QRS_NEXT_CUT()
PTP {E1 34737.351,E2 34737.351}
PTP {X 0,Y 759.916,A -85,B 0,C 180,E1 34737.351,E2 34737.351,E3 0,E4 0,E5 0,E6 0}
QRS_SPEED_INIT()
LIN {X 0,Y 759.916,Z 1215,A -85,B 0,C 180,E1 34737.351,E2 34737.351,E3 0,E4 0,E5 0,E6 0} C_VEL
LIN {X 0,Y 759.916,Z 694.953,A -85,B 0,C 180,E1 34737.351,E2 34737.351} C_VEL
LIN {X 0,Y 759.916,Z 679.951,A -85,B 0,C 180,E1 34737.351,E2 34737.351} C_VEL
LIN {X 0,Y 759.914,Z 679.08,A -85,B 0,C 180,E1 34737.064,E2 34737.064} C_VEL
LIN {X 0,Y 759.912,Z 758.546,A -85,B 0,C 180,E1 34734.185,E2 34734.185} C_VEL
LIN {X 0,Y 759.906,Z 836.117,A -85,B 0,C 180,E1 34731.411,E2 34731.411} C_VEL
LIN {X 0,Y 759.917,Z 950.864,A -85,B 0,C 180,E1 34730.313,E2 34730.313} C_VEL
LIN {X 0,Y 759.912,Z 962.666,A -85,B 0,C 180,E1 34730.113,E2 34730.113} C_VEL
LIN {X 0,Y 759.907,Z 975.52,A -85,B 0,C 180,E1 34729.789,E2 34729.789} C_VEL
LIN {X 0,Y 759.913,Z 990.031,A -85,B 0,C 180,E1 34729.27,E2 34729.27} C_VEL
LIN {X 0,Y 759.899,Z 1001.309,A -85,B 0,C 180,E1 34728.732,E2 34728.732} C_VEL
LIN {X 0,Y 759.919,Z 1011.084,A -85,B 0,C 180,E1 34728.155,E2 34728.155} C_VEL
LIN {X 0,Y 759.915,Z 1020.118,A -85,B 0,C 180,E1 34727.506,E2 34727.506} C_VEL
LIN {X 0,Y 759.915,Z 1028.572,A -85,B 0,C 180,E1 34726.765,E2 34726.765} C_VEL
LIN {X 0,Y 759.911,Z 1037.65,A -85,B 0,C 180,E1 34725.756,E2 34725.756} C_VEL
LIN {X 0,Y 759.916,Z 1043.966,A -85,B 0,C 180,E1 34724.821,E2 34724.821} C_VEL
LIN {X 0,Y 759.916,Z 1048.406,A -85,B 0,C 180,E1 34723.959,E2 34723.959} C_VEL
LIN {X 0,Y 759.912,Z 1051.646,A -85,B 0,C 180,E1 34723.095,E2 34723.095} C_VEL
LIN {X 0,Y 759.918,Z 1053.76,A -85,B 0,C 180,E1 34722.226,E2 34722.226} C_VEL
LIN {X 0,Y 759.907,Z 1054.804,A -85,B 0,C 180,E1 34721.33,E2 34721.33} C_VEL
LIN {X 0,Y 759.913,Z 1054.696,A -85,B 0,C 180,E1 34720.395,E2 34720.395} C_VEL
LIN {X 0,Y 759.905,Z 1052.996,A -85,B 0,C 180,E1 34719.271,E2 34719.271} C_VEL
LIN {X 0,Y 759.917,Z 1049.566,A -85,B 0,C 180,E1 34718.219,E2 34718.219} C_VEL
LIN {X 0,Y 759.908,Z 1045.3,A -85,B 0,C 180,E1 34717.323,E2 34717.323} C_VEL
LIN {X 0,Y 759.913,Z 1040.168,A -85,B 0,C 180,E1 34716.504,E2 34716.504} C_VEL
LIN {X 0,Y 759.917,Z 1034.354,A -85,B 0,C 180,E1 34715.761,E2 34715.761} C_VEL
LIN {X 0,Y 759.919,Z 1027.189,A -85,B 0,C 180,E1 34715.016,E2 34715.016} C_VEL
LIN {X 0,Y 759.916,Z 1019.197,A -85,B 0,C 180,E1 34714.332,E2 34714.332} C_VEL
LIN {X 0,Y 759.919,Z 1009.396,A -85,B 0,C 180,E1 34713.644,E2 34713.644} C_VEL
LIN {X 0,Y 759.904,Z 996.19,A -85,B 0,C 180,E1 34712.917,E2 34712.917} C_VEL
LIN {X 0,Y 759.914,Z 985.016,A -85,B 0,C 180,E1 34712.444,E2 34712.444} C_VEL
LIN {X 0,Y 759.906,Z 973.587,A -85,B 0,C 180,E1 34712.068,E2 34712.068} C_VEL
LIN {X 0,Y 759.914,Z 962.312,A -85,B 0,C 180,E1 34711.79,E2 34711.79} C_VEL
LIN {X 0,Y 759.916,Z 950.123,A -85,B 0,C 180,E1 34711.587,E2 34711.587} C_VEL
LIN {X 0,Y 759.905,Z 835.386,A -85,B 0,C 180,E1 34710.477,E2 34710.477} C_VEL
LIN {X 0,Y 759.917,Z 755.634,A -85,B 0,C 180,E1 34707.62,E2 34707.62} C_VEL
LIN {X 0,Y 759.913,Z 676.623,A -85,B 0,C 180,E1 34704.756,E2 34704.756} C_VEL
LIN {X 0,Y 759.914,Z 596.236,A -85,B 0,C 180,E1 34701.799,E2 34701.799} C_VEL
LIN {X 0,Y 759.89,Z 522.845,A -85,B 0,C 180,E1 34699.051,E2 34699.051} C_VEL
LIN {X 0,Y 759.918,Z 450.182,A -85,B 0,C 180,E1 34696.279,E2 34696.279} C_VEL
LIN {X 0,Y 759.918,Z 393.58,A -85,B 0,C 180,E1 34694.148,E2 34694.148} C_VEL
LIN {X 0,Y 759.86,Z 324.573,A -85,B 0,C 180,E1 34691.632,E2 34691.632} C_VEL
LIN {X 0,Y 759.869,Z 309.663,A -85,B 0,C 180,E1 34691.06,E2 34691.06} C_VEL
LIN {X 0,Y 759.887,Z 319.172,A -85,B 0,C 180,E1 34690.892,E2 34690.892} C_VEL
LIN {X 0,Y 759.917,Z 540.516,A -85,B 0,C 180,E1 34688.23,E2 34688.23} C_VEL
LIN {X 0,Y 759.912,Z 766.77,A -85,B 0,C 180,E1 34685.609,E2 34685.609} C_VEL
LIN {X 0,Y 759.911,Z 803.217,A -85,B 0,C 180,E1 34685.158,E2 34685.158} C_VEL
LIN {X 0,Y 759.908,Z 828.5,A -85,B 0,C 180,E1 34684.704,E2 34684.704} C_VEL
LIN {X 0,Y 759.915,Z 854.556,A -85,B 0,C 180,E1 34684.093,E2 34684.093} C_VEL
LIN {X 0,Y 759.906,Z 879.193,A -85,B 0,C 180,E1 34683.368,E2 34683.368} C_VEL
LIN {X 0,Y 759.918,Z 906.079,A -85,B 0,C 180,E1 34682.425,E2 34682.425} C_VEL
LIN {X 0,Y 759.915,Z 928.461,A -85,B 0,C 180,E1 34681.5,E2 34681.5} C_VEL
LIN {X 0,Y 759.914,Z 947.581,A -85,B 0,C 180,E1 34680.612,E2 34680.612} C_VEL
LIN {X 0,Y 759.914,Z 966.174,A -85,B 0,C 180,E1 34679.653,E2 34679.653} C_VEL
LIN {X 0,Y 759.91,Z 985.832,A -85,B 0,C 180,E1 34678.532,E2 34678.532} C_VEL
LIN {X 0,Y 759.91,Z 1009.761,A -85,B 0,C 180,E1 34676.998,E2 34676.998} C_VEL
LIN {X 0,Y 759.915,Z 1028.449,A -85,B 0,C 180,E1 34675.652,E2 34675.652} C_VEL
LIN {X 0,Y 759.893,Z 1047.319,A -85,B 0,C 180,E1 34674.157,E2 34674.157} C_VEL
LIN {X 0,Y 759.911,Z 1066.636,A -85,B 0,C 180,E1 34672.432,E2 34672.432} C_VEL
LIN {X 0,Y 759.897,Z 1081.386,A -85,B 0,C 180,E1 34670.972,E2 34670.972} C_VEL
LIN {X 0,Y 759.909,Z 1095.388,A -85,B 0,C 180,E1 34669.445,E2 34669.445} C_VEL
LIN {X 0,Y 759.911,Z 1111.611,A -85,B 0,C 180,E1 34667.454,E2 34667.454} C_VEL
LIN {X 0,Y 759.891,Z 1123.379,A -85,B 0,C 180,E1 34665.806,E2 34665.806} C_VEL
LIN {X 0,Y 759.916,Z 1133.313,A -85,B 0,C 180,E1 34664.245,E2 34664.245} C_VEL
LIN {X 0,Y 759.917,Z 1142.044,A -85,B 0,C 180,E1 34662.694,E2 34662.694} C_VEL
LIN {X 0,Y 759.898,Z 1149.999,A -85,B 0,C 180,E1 34661.077,E2 34661.077} C_VEL
LIN {X 0,Y 759.918,Z 1157.72,A -85,B 0,C 180,E1 34659.238,E2 34659.238} C_VEL
LIN {X 0,Y 759.912,Z 1164.34,A -85,B 0,C 180,E1 34657.258,E2 34657.258} C_VEL
LIN {X 0,Y 759.91,Z 1169.506,A -85,B 0,C 180,E1 34655.21,E2 34655.21} C_VEL
LIN {X 0,Y 759.912,Z 1173.032,A -85,B 0,C 180,E1 34653.093,E2 34653.093} C_VEL
LIN {X 0,Y 759.908,Z 1174.635,A -85,B 0,C 180,E1 34651.207,E2 34651.207} C_VEL
LIN {X 0,Y 759.89,Z 1174.841,A -85,B 0,C 180,E1 34649.398,E2 34649.398} C_VEL
LIN {X 0,Y 759.905,Z 1173.876,A -85,B 0,C 180,E1 34647.588,E2 34647.588} C_VEL
LIN {X 0,Y 759.906,Z 1171.005,A -85,B 0,C 180,E1 34645.473,E2 34645.473} C_VEL
LIN {X 0,Y 759.91,Z 1166.488,A -85,B 0,C 180,E1 34643.428,E2 34643.428} C_VEL
LIN {X 0,Y 759.917,Z 1160.522,A -85,B 0,C 180,E1 34641.45,E2 34641.45} C_VEL
LIN {X 0,Y 759.892,Z 1152.552,A -85,B 0,C 180,E1 34639.386,E2 34639.386} C_VEL
LIN {X 0,Y 759.913,Z 1142.943,A -85,B 0,C 180,E1 34637.385,E2 34637.385} C_VEL
LIN {X 0,Y 759.918,Z 1133.863,A -85,B 0,C 180,E1 34635.757,E2 34635.757} C_VEL
LIN {X 0,Y 759.897,Z 1124.515,A -85,B 0,C 180,E1 34634.274,E2 34634.274} C_VEL
LIN {X 0,Y 759.896,Z 1114.001,A -85,B 0,C 180,E1 34632.78,E2 34632.78} C_VEL
LIN {X 0,Y 759.906,Z 1101.586,A -85,B 0,C 180,E1 34631.195,E2 34631.195} C_VEL
LIN {X 0,Y 759.904,Z 1084.615,A -85,B 0,C 180,E1 34629.272,E2 34629.272} C_VEL
LIN {X 0,Y 759.894,Z 1069.306,A -85,B 0,C 180,E1 34627.732,E2 34627.732} C_VEL
LIN {X 0,Y 759.911,Z 1053.867,A -85,B 0,C 180,E1 34626.32,E2 34626.32} C_VEL
LIN {X 0,Y 759.9,Z 1033.545,A -85,B 0,C 180,E1 34624.642,E2 34624.642} C_VEL
LIN {X 0,Y 759.916,Z 1014.708,A -85,B 0,C 180,E1 34623.258,E2 34623.258} C_VEL
LIN {X 0,Y 759.901,Z 995.825,A -85,B 0,C 180,E1 34621.996,E2 34621.996} C_VEL
LIN {X 0,Y 759.904,Z 972.23,A -85,B 0,C 180,E1 34620.583,E2 34620.583} C_VEL
LIN {X 0,Y 759.915,Z 950.344,A -85,B 0,C 180,E1 34619.434,E2 34619.434} C_VEL
LIN {X 0,Y 759.912,Z 931.714,A -85,B 0,C 180,E1 34618.554,E2 34618.554} C_VEL
LIN {X 0,Y 759.919,Z 912.668,A -85,B 0,C 180,E1 34617.748,E2 34617.748} C_VEL
LIN {X 0,Y 759.92,Z 893.868,A -85,B 0,C 180,E1 34617.04,E2 34617.04} C_VEL
LIN {X 0,Y 759.909,Z 875.428,A -85,B 0,C 180,E1 34616.426,E2 34616.426} C_VEL
LIN {X 0,Y 759.912,Z 852.836,A -85,B 0,C 180,E1 34615.773,E2 34615.773} C_VEL
LIN {X 0,Y 759.914,Z 826.079,A -85,B 0,C 180,E1 34615.155,E2 34615.155} C_VEL
LIN {X 0,Y 759.91,Z 799.971,A -85,B 0,C 180,E1 34614.705,E2 34614.705} C_VEL
LIN {X 0,Y 759.919,Z 744.192,A -85,B 0,C 180,E1 34614.044,E2 34614.044} C_VEL
LIN {X 0,Y 759.912,Z 520.251,A -85,B 0,C 180,E1 34611.44,E2 34611.44} C_VEL
LIN {X 0,Y 759.881,Z 320.944,A -85,B 0,C 180,E1 34609.038,E2 34609.038} C_VEL
LIN {X 0,Y 759.906,Z 309.576,A -85,B 0,C 180,E1 34608.251,E2 34608.251} C_VEL
LIN {X 0,Y 759.906,Z 309.576,A -85,B 0,C 180,E1 34605.257,E2 34605.257} C_VEL
LIN {X 0,Y 759.897,Z 309.577,A -85,B 0,C 180,E1 34602.426,E2 34602.426} C_VEL
LIN {X 0,Y 759.915,Z 309.575,A -85,B 0,C 180,E1 34599.362,E2 34599.362} C_VEL
LIN {X 0,Y 759.895,Z 309.577,A -85,B 0,C 180,E1 34596.589,E2 34596.589} C_VEL
LIN {X 0,Y 759.894,Z 309.575,A -85,B 0,C 180,E1 34593.73,E2 34593.73} C_VEL
LIN {X 0,Y 759.909,Z 309.577,A -85,B 0,C 180,E1 34590.875,E2 34590.875} C_VEL
LIN {X 0,Y 759.88,Z 309.577,A -85,B 0,C 180,E1 34588.104,E2 34588.104} C_VEL
LIN {X 0,Y 759.916,Z 309.575,A -85,B 0,C 180,E1 34585.234,E2 34585.234} C_VEL
LIN {X 0,Y 759.888,Z 309.577,A -85,B 0,C 180,E1 34582.433,E2 34582.433} C_VEL
LIN {X 0,Y 759.881,Z 309.576,A -85,B 0,C 180,E1 34579.766,E2 34579.766} C_VEL
LIN {X 0,Y 759.919,Z 309.577,A -85,B 0,C 180,E1 34576.905,E2 34576.905} C_VEL
LIN {X 0,Y 759.88,Z 309.577,A -85,B 0,C 180,E1 34574.012,E2 34574.012} C_VEL
LIN {X 0,Y 759.899,Z 309.577,A -85,B 0,C 180,E1 34571.23,E2 34571.23} C_VEL
LIN {X 0,Y 759.889,Z 309.577,A -85,B 0,C 180,E1 34568.399,E2 34568.399} C_VEL
LIN {X 0,Y 759.884,Z 309.576,A -85,B 0,C 180,E1 34565.588,E2 34565.588} C_VEL
LIN {X 0,Y 759.919,Z 309.576,A -85,B 0,C 180,E1 34562.791,E2 34562.791} C_VEL
LIN {X 0,Y 759.881,Z 309.577,A -85,B 0,C 180,E1 34559.849,E2 34559.849} C_VEL
LIN {X 0,Y 759.913,Z 309.576,A -85,B 0,C 180,E1 34557.03,E2 34557.03} C_VEL
LIN {X 0,Y 759.903,Z 309.574,A -85,B 0,C 180,E1 34554.109,E2 34554.109} C_VEL
LIN {X 0,Y 759.91,Z 309.578,A -85,B 0,C 180,E1 34551.144,E2 34551.144} C_VEL
LIN {X 0,Y 759.916,Z 309.572,A -85,B 0,C 180,E1 34548.155,E2 34548.155} C_VEL
LIN {X 0,Y 759.912,Z 309.576,A -85,B 0,C 180,E1 34545.211,E2 34545.211} C_VEL
LIN {X 0,Y 759.898,Z 309.574,A -85,B 0,C 180,E1 34542.293,E2 34542.293} C_VEL
LIN {X 0,Y 759.917,Z 309.575,A -85,B 0,C 180,E1 34539.432,E2 34539.432} C_VEL
LIN {X 0,Y 759.882,Z 309.576,A -85,B 0,C 180,E1 34536.605,E2 34536.605} C_VEL
LIN {X 0,Y 759.905,Z 337.086,A -85,B 0,C 180,E1 34534.557,E2 34534.557} C_VEL
LIN {X 0,Y 759.898,Z 371.805,A -85,B 0,C 180,E1 34532.11,E2 34532.11} C_VEL
LIN {X 0,Y 759.915,Z 409.049,A -85,B 0,C 180,E1 34529.607,E2 34529.607} C_VEL
LIN {X 0,Y 759.914,Z 451.966,A -85,B 0,C 180,E1 34526.858,E2 34526.858} C_VEL
LIN {X 0,Y 759.917,Z 494.443,A -85,B 0,C 180,E1 34524.253,E2 34524.253} C_VEL
LIN {X 0,Y 759.917,Z 511.943,A -85,B 0,C 180,E1 34523.177,E2 34523.177} C_VEL
LIN {X 0,Y 759.868,Z 518.357,A -85,B 0,C 180,E1 34522.632,E2 34522.632} C_VEL
LIN {X 0,Y 759.872,Z 521.733,A -85,B 0,C 180,E1 34522.179,E2 34522.179} C_VEL
LIN {X 0,Y 759.916,Z 522.967,A -85,B 0,C 180,E1 34521.767,E2 34521.767} C_VEL
LIN {X 0,Y 759.913,Z 522.331,A -85,B 0,C 180,E1 34521.414,E2 34521.414} C_VEL
LIN {X 0,Y 759.893,Z 519.98,A -85,B 0,C 180,E1 34521.123,E2 34521.123} C_VEL
LIN {X 0,Y 759.887,Z 515.523,A -85,B 0,C 180,E1 34520.878,E2 34520.878} C_VEL
LIN {X 0,Y 759.891,Z 508.959,A -85,B 0,C 180,E1 34520.71,E2 34520.71} C_VEL
LIN {X 0,Y 759.895,Z 499.107,A -85,B 0,C 180,E1 34520.633,E2 34520.633} C_VEL
LIN {X 0,Y 759.896,Z 309.577,A -85,B 0,C 180,E1 34520.619,E2 34520.619} C_VEL
LIN {X 0,Y 759.885,Z 309.578,A -85,B 0,C 180,E1 34517.849,E2 34517.849} C_VEL
LIN {X 0,Y 759.914,Z 309.575,A -85,B 0,C 180,E1 34515.042,E2 34515.042} C_VEL
LIN {X 0,Y 759.901,Z 309.831,A -85,B 0,C 180,E1 34513.53,E2 34513.53} C_VEL
LIN {X 0,Y 759.904,Z 350.586,A -85,B 0,C 180,E1 34510.919,E2 34510.919} C_VEL
LIN {X 0,Y 759.912,Z 566.45,A -85,B 0,C 180,E1 34508.323,E2 34508.323} C_VEL
LIN {X 0,Y 759.917,Z 792.192,A -85,B 0,C 180,E1 34505.706,E2 34505.706} C_VEL
LIN {X 0,Y 759.911,Z 831.842,A -85,B 0,C 180,E1 34505.223,E2 34505.223} C_VEL
LIN {X 0,Y 759.908,Z 857.533,A -85,B 0,C 180,E1 34504.769,E2 34504.769} C_VEL
LIN {X 0,Y 759.913,Z 884.387,A -85,B 0,C 180,E1 34504.143,E2 34504.143} C_VEL
LIN {X 0,Y 759.907,Z 909.999,A -85,B 0,C 180,E1 34503.388,E2 34503.388} C_VEL
LIN {X 0,Y 759.918,Z 937.266,A -85,B 0,C 180,E1 34502.422,E2 34502.422} C_VEL
LIN {X 0,Y 759.915,Z 958.597,A -85,B 0,C 180,E1 34501.539,E2 34501.539} C_VEL
LIN {X 0,Y 759.912,Z 977.517,A -85,B 0,C 180,E1 34500.66,E2 34500.66} C_VEL
LIN {X 0,Y 759.912,Z 996.378,A -85,B 0,C 180,E1 34499.687,E2 34499.687} C_VEL
LIN {X 0,Y 759.903,Z 1015.171,A -85,B 0,C 180,E1 34498.616,E2 34498.616} C_VEL
LIN {X 0,Y 759.901,Z 1038.015,A -85,B 0,C 180,E1 34497.166,E2 34497.166} C_VEL
LIN {X 0,Y 759.916,Z 1057.965,A -85,B 0,C 180,E1 34495.734,E2 34495.734} C_VEL
LIN {X 0,Y 759.902,Z 1075.357,A -85,B 0,C 180,E1 34494.361,E2 34494.361} C_VEL
LIN {X 0,Y 759.914,Z 1095.42,A -85,B 0,C 180,E1 34492.593,E2 34492.593} C_VEL
LIN {X 0,Y 759.892,Z 1110.551,A -85,B 0,C 180,E1 34491.104,E2 34491.104} C_VEL
LIN {X 0,Y 759.911,Z 1124.385,A -85,B 0,C 180,E1 34489.603,E2 34489.603} C_VEL
LIN {X 0,Y 759.914,Z 1139.588,A -85,B 0,C 180,E1 34487.773,E2 34487.773} C_VEL
LIN {X 0,Y 759.889,Z 1152.649,A -85,B 0,C 180,E1 34485.961,E2 34485.961} C_VEL
LIN {X 0,Y 759.91,Z 1162.664,A -85,B 0,C 180,E1 34484.399,E2 34484.399} C_VEL
LIN {X 0,Y 759.914,Z 1171.531,A -85,B 0,C 180,E1 34482.836,E2 34482.836} C_VEL
LIN {X 0,Y 759.915,Z 1179.146,A -85,B 0,C 180,E1 34481.305,E2 34481.305} C_VEL
LIN {X 0,Y 759.906,Z 1186.727,A -85,B 0,C 180,E1 34479.542,E2 34479.542} C_VEL
LIN {X 0,Y 759.908,Z 1193.596,A -85,B 0,C 180,E1 34477.56,E2 34477.56} C_VEL
LIN {X 0,Y 759.91,Z 1199.11,A -85,B 0,C 180,E1 34475.435,E2 34475.435} C_VEL
LIN {X 0,Y 759.916,Z 1202.587,A -85,B 0,C 180,E1 34473.469,E2 34473.469} C_VEL
LIN {X 0,Y 759.914,Z 1204.581,A -85,B 0,C 180,E1 34471.432,E2 34471.432} C_VEL
LIN {X 0,Y 759.889,Z 1204.849,A -85,B 0,C 180,E1 34469.471,E2 34469.471} C_VEL
LIN {X 0,Y 759.907,Z 1203.906,A -85,B 0,C 180,E1 34467.661,E2 34467.661} C_VEL
LIN {X 0,Y 759.908,Z 1201.052,A -85,B 0,C 180,E1 34465.547,E2 34465.547} C_VEL
LIN {X 0,Y 759.914,Z 1196.563,A -85,B 0,C 180,E1 34463.502,E2 34463.502} C_VEL
LIN {X 0,Y 759.912,Z 1190.625,A -85,B 0,C 180,E1 34461.525,E2 34461.525} C_VEL
LIN {X 0,Y 759.896,Z 1182.676,A -85,B 0,C 180,E1 34459.461,E2 34459.461} C_VEL
LIN {X 0,Y 759.905,Z 1173.105,A -85,B 0,C 180,E1 34457.46,E2 34457.46} C_VEL
LIN {X 0,Y 759.91,Z 1164.049,A -85,B 0,C 180,E1 34455.833,E2 34455.833} C_VEL
LIN {X 0,Y 759.894,Z 1154.204,A -85,B 0,C 180,E1 34454.272,E2 34454.272} C_VEL
LIN {X 0,Y 759.904,Z 1143.658,A -85,B 0,C 180,E1 34452.778,E2 34452.778} C_VEL
LIN {X 0,Y 759.896,Z 1129.919,A -85,B 0,C 180,E1 34451.033,E2 34451.033} C_VEL
LIN {X 0,Y 759.898,Z 1113.38,A -85,B 0,C 180,E1 34449.189,E2 34449.189} C_VEL
LIN {X 0,Y 759.898,Z 1098.813,A -85,B 0,C 180,E1 34447.73,E2 34447.73} C_VEL
LIN {X 0,Y 759.911,Z 1082.64,A -85,B 0,C 180,E1 34446.256,E2 34446.256} C_VEL
LIN {X 0,Y 759.91,Z 1061.259,A -85,B 0,C 180,E1 34444.515,E2 34444.515} C_VEL
LIN {X 0,Y 759.909,Z 1043.428,A -85,B 0,C 180,E1 34443.213,E2 34443.213} C_VEL
LIN {X 0,Y 759.914,Z 1024.236,A -85,B 0,C 180,E1 34441.939,E2 34441.939} C_VEL
LIN {X 0,Y 759.906,Z 999.416,A -85,B 0,C 180,E1 34440.477,E2 34440.477} C_VEL
LIN {X 0,Y 759.913,Z 979.389,A -85,B 0,C 180,E1 34439.432,E2 34439.432} C_VEL
LIN {X 0,Y 759.912,Z 960.652,A -85,B 0,C 180,E1 34438.552,E2 34438.552} C_VEL
LIN {X 0,Y 759.918,Z 941.519,A -85,B 0,C 180,E1 34437.747,E2 34437.747} C_VEL
LIN {X 0,Y 759.92,Z 922.548,A -85,B 0,C 180,E1 34437.038,E2 34437.038} C_VEL
LIN {X 0,Y 759.91,Z 903.935,A -85,B 0,C 180,E1 34436.425,E2 34436.425} C_VEL
LIN {X 0,Y 759.914,Z 881.874,A -85,B 0,C 180,E1 34435.793,E2 34435.793} C_VEL
LIN {X 0,Y 759.909,Z 855.665,A -85,B 0,C 180,E1 34435.192,E2 34435.192} C_VEL
LIN {X 0,Y 759.91,Z 828.993,A -85,B 0,C 180,E1 34434.735,E2 34434.735} C_VEL
LIN {X 0,Y 759.914,Z 731.51,A -85,B 0,C 180,E1 34433.599,E2 34433.599} C_VEL
LIN {X 0,Y 759.915,Z 508.586,A -85,B 0,C 180,E1 34430.991,E2 34430.991} C_VEL
LIN {X 0,Y 759.916,Z 343.629,A -85,B 0,C 180,E1 34428.982,E2 34428.982} C_VEL
LIN {X 0,Y 759.896,Z 309.576,A -85,B 0,C 180,E1 34428.331,E2 34428.331} C_VEL
LIN {X 0,Y 759.903,Z 309.578,A -85,B 0,C 180,E1 34425.494,E2 34425.494} C_VEL
LIN {X 0,Y 759.909,Z 309.577,A -85,B 0,C 180,E1 34422.647,E2 34422.647} C_VEL
LIN {X 0,Y 759.877,Z 309.577,A -85,B 0,C 180,E1 34419.784,E2 34419.784} C_VEL
LIN {X 0,Y 759.883,Z 309.574,A -85,B 0,C 180,E1 34417.061,E2 34417.061} C_VEL
LIN {X 0,Y 759.907,Z 309.575,A -85,B 0,C 180,E1 34414.093,E2 34414.093} C_VEL
LIN {X 0,Y 759.918,Z 309.575,A -85,B 0,C 180,E1 34411.211,E2 34411.211} C_VEL
LIN {X 0,Y 759.919,Z 309.573,A -85,B 0,C 180,E1 34408.274,E2 34408.274} C_VEL
LIN {X 0,Y 759.873,Z 309.575,A -85,B 0,C 180,E1 34405.311,E2 34405.311} C_VEL
LIN {X 0,Y 759.875,Z 309.577,A -85,B 0,C 180,E1 34402.678,E2 34402.678} C_VEL
LIN {X 0,Y 759.914,Z 309.574,A -85,B 0,C 180,E1 34399.815,E2 34399.815} C_VEL
LIN {X 0,Y 759.907,Z 309.577,A -85,B 0,C 180,E1 34396.944,E2 34396.944} C_VEL
LIN {X 0,Y 759.913,Z 309.573,A -85,B 0,C 180,E1 34394.011,E2 34394.011} C_VEL
LIN {X 0,Y 759.881,Z 309.577,A -85,B 0,C 180,E1 34390.999,E2 34390.999} C_VEL
LIN {X 0,Y 759.916,Z 309.801,A -85,B 0,C 180,E1 34390.594,E2 34390.594} C_VEL
LIN {X 0,Y 759.917,Z 389.194,A -85,B 0,C 180,E1 34387.865,E2 34387.865} C_VEL
LIN {X 0,Y 759.904,Z 437.584,A -85,B 0,C 180,E1 34386.118,E2 34386.118} C_VEL
LIN {X 0,Y 759.914,Z 512.66,A -85,B 0,C 180,E1 34383.243,E2 34383.243} C_VEL
LIN {X 0,Y 759.891,Z 587.07,A -85,B 0,C 180,E1 34380.452,E2 34380.452} C_VEL
LIN {X 0,Y 759.911,Z 661.684,A -85,B 0,C 180,E1 34377.7,E2 34377.7} C_VEL
LIN {X 0,Y 759.914,Z 679.08,A -85,B 0,C 180,E1 34377.064,E2 34377.064} C_VEL
LIN {X 0,Y 758.952,Z 686.122,A -85,B 0,C 180,E1 34376.828,E2 34376.828} C_VEL
LIN {X 0,Y 752.87,Z 705.08,A -85,B 0,C 180,E1 34376.263,E2 34376.263} C_VEL
LIN {X 0,Y 752.141,Z 711.123,A -85,B 0,C 180,E1 34376.057,E2 34376.057} C_VEL
LIN {X 0,Y 752.048,Z 789.43,A -85,B 0,C 180,E1 34373.204,E2 34373.204} C_VEL
LIN {X 0,Y 752.039,Z 836.739,A -85,B 0,C 180,E1 34371.516,E2 34371.516} C_VEL
LIN {X 0,Y 752.023,Z 951.389,A -85,B 0,C 180,E1 34370.406,E2 34370.406} C_VEL
LIN {X 0,Y 752.007,Z 965.681,A -85,B 0,C 180,E1 34370.149,E2 34370.149} C_VEL
LIN {X 0,Y 751.99,Z 980.545,A -85,B 0,C 180,E1 34369.72,E2 34369.72} C_VEL
LIN {X 0,Y 751.975,Z 992.811,A -85,B 0,C 180,E1 34369.233,E2 34369.233} C_VEL
LIN {X 0,Y 751.954,Z 1003.593,A -85,B 0,C 180,E1 34368.689,E2 34368.689} C_VEL
LIN {X 0,Y 751.952,Z 1014.743,A -85,B 0,C 180,E1 34367.989,E2 34367.989} C_VEL
LIN {X 0,Y 751.934,Z 1024.967,A -85,B 0,C 180,E1 34367.169,E2 34367.169} C_VEL
LIN {X 0,Y 751.928,Z 1033.456,A -85,B 0,C 180,E1 34366.308,E2 34366.308} C_VEL
LIN {X 0,Y 751.922,Z 1039.959,A -85,B 0,C 180,E1 34365.485,E2 34365.485} C_VEL
LIN {X 0,Y 751.912,Z 1045.589,A -85,B 0,C 180,E1 34364.576,E2 34364.576} C_VEL
LIN {X 0,Y 751.912,Z 1050.595,A -85,B 0,C 180,E1 34363.466,E2 34363.466} C_VEL
LIN {X 0,Y 751.915,Z 1053.568,A -85,B 0,C 180,E1 34362.35,E2 34362.35} C_VEL
LIN {X 0,Y 751.908,Z 1054.774,A -85,B 0,C 180,E1 34361.388,E2 34361.388} C_VEL
LIN {X 0,Y 751.912,Z 1054.715,A -85,B 0,C 180,E1 34360.421,E2 34360.421} C_VEL
LIN {X 0,Y 751.906,Z 1053.069,A -85,B 0,C 180,E1 34359.284,E2 34359.284} C_VEL
LIN {X 0,Y 751.917,Z 1049.358,A -85,B 0,C 180,E1 34358.14,E2 34358.14} C_VEL
LIN {X 0,Y 751.913,Z 1045.023,A -85,B 0,C 180,E1 34357.234,E2 34357.234} C_VEL
LIN {X 0,Y 751.923,Z 1039.63,A -85,B 0,C 180,E1 34356.379,E2 34356.379} C_VEL
LIN {X 0,Y 751.926,Z 1033.188,A -85,B 0,C 180,E1 34355.571,E2 34355.571} C_VEL
LIN {X 0,Y 751.939,Z 1024.748,A -85,B 0,C 180,E1 34354.72,E2 34354.72} C_VEL
LIN {X 0,Y 751.955,Z 1013.524,A -85,B 0,C 180,E1 34353.84,E2 34353.84} C_VEL
LIN {X 0,Y 751.951,Z 1003.326,A -85,B 0,C 180,E1 34353.206,E2 34353.206} C_VEL
LIN {X 0,Y 751.976,Z 992.248,A -85,B 0,C 180,E1 34352.652,E2 34352.652} C_VEL
LIN {X 0,Y 751.987,Z 979.149,A -85,B 0,C 180,E1 34352.14,E2 34352.14} C_VEL
LIN {X 0,Y 752.01,Z 963.946,A -85,B 0,C 180,E1 34351.726,E2 34351.726} C_VEL
LIN {X 0,Y 752.022,Z 950.66,A -85,B 0,C 180,E1 34351.494,E2 34351.494} C_VEL
LIN {X 0,Y 752.016,Z 835.782,A -85,B 0,C 180,E1 34350.38,E2 34350.38} C_VEL
LIN {X 0,Y 752.096,Z 755.202,A -85,B 0,C 180,E1 34347.463,E2 34347.463} C_VEL
LIN {X 0,Y 752.178,Z 675.878,A -85,B 0,C 180,E1 34344.557,E2 34344.557} C_VEL
LIN {X 0,Y 752.281,Z 596.524,A -85,B 0,C 180,E1 34341.607,E2 34341.607} C_VEL
LIN {X 0,Y 752.373,Z 521.834,A -85,B 0,C 180,E1 34338.782,E2 34338.782} C_VEL
LIN {X 0,Y 752.428,Z 453.896,A -85,B 0,C 180,E1 34336.183,E2 34336.183} C_VEL
LIN {X 0,Y 752.292,Z 406.665,A -85,B 0,C 180,E1 34334.414,E2 34334.414} C_VEL
LIN {X 0,Y 752.341,Z 331.817,A -85,B 0,C 180,E1 34331.675,E2 34331.675} C_VEL
LIN {X 0,Y 752.372,Z 323.165,A -85,B 0,C 180,E1 34331.341,E2 34331.341} C_VEL
LIN {X 0,Y 753.749,Z 325.279,A -85,B 0,C 180,E1 34331.222,E2 34331.222} C_VEL
LIN {X 0,Y 753.655,Z 505.38,A -85,B 0,C 180,E1 34329.028,E2 34329.028} C_VEL
LIN {X 0,Y 753.438,Z 733.72,A -85,B 0,C 180,E1 34326.345,E2 34326.345} C_VEL
LIN {X 0,Y 753.352,Z 799.65,A -85,B 0,C 180,E1 34325.563,E2 34325.563} C_VEL
LIN {X 0,Y 753.277,Z 826.497,A -85,B 0,C 180,E1 34325.098,E2 34325.098} C_VEL
LIN {X 0,Y 753.193,Z 854.407,A -85,B 0,C 180,E1 34324.444,E2 34324.444} C_VEL
LIN {X 0,Y 753.094,Z 878.412,A -85,B 0,C 180,E1 34323.735,E2 34323.735} C_VEL
LIN {X 0,Y 752.988,Z 903.865,A -85,B 0,C 180,E1 34322.851,E2 34322.851} C_VEL
LIN {X 0,Y 752.861,Z 927.675,A -85,B 0,C 180,E1 34321.866,E2 34321.866} C_VEL
LIN {X 0,Y 752.761,Z 947.599,A -85,B 0,C 180,E1 34320.935,E2 34320.935} C_VEL
LIN {X 0,Y 752.666,Z 966.993,A -85,B 0,C 180,E1 34319.924,E2 34319.924} C_VEL
LIN {X 0,Y 752.563,Z 987.659,A -85,B 0,C 180,E1 34318.728,E2 34318.728} C_VEL
LIN {X 0,Y 752.423,Z 1010.984,A -85,B 0,C 180,E1 34317.203,E2 34317.203} C_VEL
LIN {X 0,Y 752.347,Z 1029.569,A -85,B 0,C 180,E1 34315.845,E2 34315.845} C_VEL
LIN {X 0,Y 752.234,Z 1049.49,A -85,B 0,C 180,E1 34314.237,E2 34314.237} C_VEL
LIN {X 0,Y 752.171,Z 1067.498,A -85,B 0,C 180,E1 34312.593,E2 34312.593} C_VEL
LIN {X 0,Y 752.096,Z 1082.173,A -85,B 0,C 180,E1 34311.118,E2 34311.118} C_VEL
LIN {X 0,Y 752.054,Z 1098.235,A -85,B 0,C 180,E1 34309.334,E2 34309.334} C_VEL
LIN {X 0,Y 752.003,Z 1112.745,A -85,B 0,C 180,E1 34307.488,E2 34307.488} C_VEL
LIN {X 0,Y 751.955,Z 1123.417,A -85,B 0,C 180,E1 34305.973,E2 34305.973} C_VEL
LIN {X 0,Y 751.959,Z 1133.317,A -85,B 0,C 180,E1 34304.399,E2 34304.399} C_VEL
LIN {X 0,Y 751.932,Z 1142.047,A -85,B 0,C 180,E1 34302.831,E2 34302.831} C_VEL
LIN {X 0,Y 751.923,Z 1150.002,A -85,B 0,C 180,E1 34301.196,E2 34301.196} C_VEL
LIN {X 0,Y 751.926,Z 1158.014,A -85,B 0,C 180,E1 34299.26,E2 34299.26} C_VEL
LIN {X 0,Y 751.916,Z 1164.617,A -85,B 0,C 180,E1 34297.239,E2 34297.239} C_VEL
LIN {X 0,Y 751.907,Z 1169.505,A -85,B 0,C 180,E1 34295.266,E2 34295.266} C_VEL
LIN {X 0,Y 751.911,Z 1172.929,A -85,B 0,C 180,E1 34293.203,E2 34293.203} C_VEL
LIN {X 0,Y 751.911,Z 1174.615,A -85,B 0,C 180,E1 34291.296,E2 34291.296} C_VEL
LIN {X 0,Y 751.889,Z 1174.866,A -85,B 0,C 180,E1 34289.468,E2 34289.468} C_VEL
LIN {X 0,Y 751.907,Z 1173.955,A -85,B 0,C 180,E1 34287.638,E2 34287.638} C_VEL
LIN {X 0,Y 751.908,Z 1171.13,A -85,B 0,C 180,E1 34285.501,E2 34285.501} C_VEL
LIN {X 0,Y 751.917,Z 1166.876,A -85,B 0,C 180,E1 34283.511,E2 34283.511} C_VEL
LIN {X 0,Y 751.924,Z 1160.79,A -85,B 0,C 180,E1 34281.436,E2 34281.436} C_VEL
LIN {X 0,Y 751.905,Z 1152.822,A -85,B 0,C 180,E1 34279.338,E2 34279.338} C_VEL
LIN {X 0,Y 751.941,Z 1143.351,A -85,B 0,C 180,E1 34277.327,E2 34277.327} C_VEL
LIN {X 0,Y 751.961,Z 1134.326,A -85,B 0,C 180,E1 34275.682,E2 34275.682} C_VEL
LIN {X 0,Y 751.956,Z 1124.511,A -85,B 0,C 180,E1 34274.103,E2 34274.103} C_VEL
LIN {X 0,Y 751.997,Z 1113.998,A -85,B 0,C 180,E1 34272.593,E2 34272.593} C_VEL
LIN {X 0,Y 752.031,Z 1101.583,A -85,B 0,C 180,E1 34270.99,E2 34270.99} C_VEL
LIN {X 0,Y 752.09,Z 1084.612,A -85,B 0,C 180,E1 34269.047,E2 34269.047} C_VEL
LIN {X 0,Y 752.152,Z 1069.304,A -85,B 0,C 180,E1 34267.491,E2 34267.491} C_VEL
LIN {X 0,Y 752.21,Z 1052.646,A -85,B 0,C 180,E1 34265.953,E2 34265.953} C_VEL
LIN {X 0,Y 752.343,Z 1031.328,A -85,B 0,C 180,E1 34264.2,E2 34264.2} C_VEL
LIN {X 0,Y 752.415,Z 1012.89,A -85,B 0,C 180,E1 34262.841,E2 34262.841} C_VEL
LIN {X 0,Y 752.546,Z 990.973,A -85,B 0,C 180,E1 34261.382,E2 34261.382} C_VEL
LIN {X 0,Y 752.657,Z 968.678,A -85,B 0,C 180,E1 34260.078,E2 34260.078} C_VEL
LIN {X 0,Y 752.758,Z 949.448,A -85,B 0,C 180,E1 34259.067,E2 34259.067} C_VEL
LIN {X 0,Y 752.853,Z 929.72,A -85,B 0,C 180,E1 34258.136,E2 34258.136} C_VEL
LIN {X 0,Y 752.951,Z 909.498,A -85,B 0,C 180,E1 34257.285,E2 34257.285} C_VEL
LIN {X 0,Y 753.076,Z 884.196,A -85,B 0,C 180,E1 34256.356,E2 34256.356} C_VEL
LIN {X 0,Y 753.178,Z 856.109,A -85,B 0,C 180,E1 34255.512,E2 34255.512} C_VEL
LIN {X 0,Y 753.274,Z 830.147,A -85,B 0,C 180,E1 34254.89,E2 34254.89} C_VEL
LIN {X 0,Y 753.349,Z 803.571,A -85,B 0,C 180,E1 34254.404,E2 34254.404} C_VEL
LIN {X 0,Y 753.404,Z 766.162,A -85,B 0,C 180,E1 34253.938,E2 34253.938} C_VEL
LIN {X 0,Y 753.622,Z 541.107,A -85,B 0,C 180,E1 34251.308,E2 34251.308} C_VEL
LIN {X 0,Y 753.807,Z 332.716,A -85,B 0,C 180,E1 34248.784,E2 34248.784} C_VEL
LIN {X 0,Y 753.616,Z 322.593,A -85,B 0,C 180,E1 34248.646,E2 34248.646} C_VEL
LIN {X 0,Y 753.197,Z 320.525,A -85,B 0,C 180,E1 34248.567,E2 34248.567} C_VEL
LIN {X 0,Y 753.124,Z 313.818,A -85,B 0,C 180,E1 34248.104,E2 34248.104} C_VEL
LIN {X 0,Y 751.976,Z 310.564,A -85,B 0,C 180,E1 34247.786,E2 34247.786} C_VEL
LIN {X 0,Y 751.964,Z 310.566,A -85,B 0,C 180,E1 34244.87,E2 34244.87} C_VEL
LIN {X 0,Y 751.955,Z 310.565,A -85,B 0,C 180,E1 34241.979,E2 34241.979} C_VEL
LIN {X 0,Y 751.972,Z 310.567,A -85,B 0,C 180,E1 34239.169,E2 34239.169} C_VEL
LIN {X 0,Y 751.944,Z 310.566,A -85,B 0,C 180,E1 34236.375,E2 34236.375} C_VEL
LIN {X 0,Y 751.979,Z 310.562,A -85,B 0,C 180,E1 34233.401,E2 34233.401} C_VEL
LIN {X 0,Y 751.943,Z 310.566,A -85,B 0,C 180,E1 34230.499,E2 34230.499} C_VEL
LIN {X 0,Y 751.952,Z 310.566,A -85,B 0,C 180,E1 34227.737,E2 34227.737} C_VEL
LIN {X 0,Y 751.961,Z 310.563,A -85,B 0,C 180,E1 34224.929,E2 34224.929} C_VEL
LIN {X 0,Y 751.942,Z 310.566,A -85,B 0,C 180,E1 34222.106,E2 34222.106} C_VEL
LIN {X 0,Y 751.977,Z 310.564,A -85,B 0,C 180,E1 34219.254,E2 34219.254} C_VEL
LIN {X 0,Y 751.942,Z 310.565,A -85,B 0,C 180,E1 34216.374,E2 34216.374} C_VEL
LIN {X 0,Y 751.958,Z 310.566,A -85,B 0,C 180,E1 34213.593,E2 34213.593} C_VEL
LIN {X 0,Y 751.972,Z 310.56,A -85,B 0,C 180,E1 34210.701,E2 34210.701} C_VEL
LIN {X 0,Y 751.96,Z 310.566,A -85,B 0,C 180,E1 34207.718,E2 34207.718} C_VEL
LIN {X 0,Y 751.972,Z 310.563,A -85,B 0,C 180,E1 34204.882,E2 34204.882} C_VEL
LIN {X 0,Y 751.968,Z 310.564,A -85,B 0,C 180,E1 34201.829,E2 34201.829} C_VEL
LIN {X 0,Y 751.959,Z 310.565,A -85,B 0,C 180,E1 34199.01,E2 34199.01} C_VEL
LIN {X 0,Y 751.974,Z 310.564,A -85,B 0,C 180,E1 34195.959,E2 34195.959} C_VEL
LIN {X 0,Y 751.948,Z 310.563,A -85,B 0,C 180,E1 34193.127,E2 34193.127} C_VEL
LIN {X 0,Y 751.979,Z 310.564,A -85,B 0,C 180,E1 34190.123,E2 34190.123} C_VEL
LIN {X 0,Y 751.947,Z 310.566,A -85,B 0,C 180,E1 34187.248,E2 34187.248} C_VEL
LIN {X 0,Y 751.95,Z 310.565,A -85,B 0,C 180,E1 34184.419,E2 34184.419} C_VEL
LIN {X 0,Y 751.965,Z 310.562,A -85,B 0,C 180,E1 34181.631,E2 34181.631} C_VEL
LIN {X 0,Y 751.941,Z 310.559,A -85,B 0,C 180,E1 34178.878,E2 34178.878} C_VEL
LIN {X 0,Y 751.982,Z 310.698,A -85,B 0,C 180,E1 34177.298,E2 34177.298} C_VEL
LIN {X 0,Y 753.452,Z 314.314,A -85,B 0,C 180,E1 34176.87,E2 34176.87} C_VEL
LIN {X 0,Y 753.991,Z 315.541,A -85,B 0,C 180,E1 34176.722,E2 34176.722} C_VEL
LIN {X 0,Y 753.854,Z 350.068,A -85,B 0,C 180,E1 34174.169,E2 34174.169} C_VEL
LIN {X 0,Y 753.669,Z 386.146,A -85,B 0,C 180,E1 34171.643,E2 34171.643} C_VEL
LIN {X 0,Y 753.52,Z 423.458,A -85,B 0,C 180,E1 34169.15,E2 34169.15} C_VEL
LIN {X 0,Y 753.355,Z 463.415,A -85,B 0,C 180,E1 34166.596,E2 34166.596} C_VEL
LIN {X 0,Y 753.19,Z 504.535,A -85,B 0,C 180,E1 34164.071,E2 34164.071} C_VEL
LIN {X 0,Y 753.684,Z 519.279,A -85,B 0,C 180,E1 34163.155,E2 34163.155} C_VEL
LIN {X 0,Y 754.617,Z 525.354,A -85,B 0,C 180,E1 34162.654,E2 34162.654} C_VEL
LIN {X 0,Y 755.49,Z 528.726,A -85,B 0,C 180,E1 34162.195,E2 34162.195} C_VEL
LIN {X 0,Y 756.192,Z 530.054,A -85,B 0,C 180,E1 34161.758,E2 34161.758} C_VEL
LIN {X 0,Y 756.552,Z 529.669,A -85,B 0,C 180,E1 34161.358,E2 34161.358} C_VEL
LIN {X 0,Y 756.531,Z 527.732,A -85,B 0,C 180,E1 34160.997,E2 34160.997} C_VEL
LIN {X 0,Y 756.116,Z 524.026,A -85,B 0,C 180,E1 34160.676,E2 34160.676} C_VEL
LIN {X 0,Y 755.39,Z 518.66,A -85,B 0,C 180,E1 34160.437,E2 34160.437} C_VEL
LIN {X 0,Y 754.465,Z 511.327,A -85,B 0,C 180,E1 34160.295,E2 34160.295} C_VEL
LIN {X 0,Y 753.733,Z 499.366,A -85,B 0,C 180,E1 34160.247,E2 34160.247} C_VEL
LIN {X 0,Y 753.592,Z 314.488,A -85,B 0,C 180,E1 34160.238,E2 34160.238} C_VEL
LIN {X 0,Y 752.08,Z 311.265,A -85,B 0,C 180,E1 34160.142,E2 34160.142} C_VEL
LIN {X 0,Y 751.961,Z 310.566,A -85,B 0,C 180,E1 34160.134,E2 34160.134} C_VEL
LIN {X 0,Y 751.969,Z 310.563,A -85,B 0,C 180,E1 34157.22,E2 34157.22} C_VEL
LIN {X 0,Y 751.931,Z 310.569,A -85,B 0,C 180,E1 34154.323,E2 34154.323} C_VEL
LIN {X 0,Y 751.959,Z 310.809,A -85,B 0,C 180,E1 34154.042,E2 34154.042} C_VEL
LIN {X 0,Y 753.413,Z 314.771,A -85,B 0,C 180,E1 34153.672,E2 34153.672} C_VEL
LIN {X 0,Y 753.396,Z 351.09,A -85,B 0,C 180,E1 34151.343,E2 34151.343} C_VEL
LIN {X 0,Y 753.838,Z 354.185,A -85,B 0,C 180,E1 34151.275,E2 34151.275} C_VEL
LIN {X 0,Y 753.62,Z 569.225,A -85,B 0,C 180,E1 34148.669,E2 34148.669} C_VEL
LIN {X 0,Y 753.408,Z 794.311,A -85,B 0,C 180,E1 34146.038,E2 34146.038} C_VEL
LIN {X 0,Y 753.35,Z 832.658,A -85,B 0,C 180,E1 34145.564,E2 34145.564} C_VEL
LIN {X 0,Y 753.271,Z 858.411,A -85,B 0,C 180,E1 34145.102,E2 34145.102} C_VEL
LIN {X 0,Y 753.186,Z 885.287,A -85,B 0,C 180,E1 34144.466,E2 34144.466} C_VEL
LIN {X 0,Y 753.087,Z 912.764,A -85,B 0,C 180,E1 34143.645,E2 34143.645} C_VEL
LIN {X 0,Y 752.954,Z 938.394,A -85,B 0,C 180,E1 34142.715,E2 34142.715} C_VEL
LIN {X 0,Y 752.856,Z 958.719,A -85,B 0,C 180,E1 34141.864,E2 34141.864} C_VEL
LIN {X 0,Y 752.757,Z 978.551,A -85,B 0,C 180,E1 34140.933,E2 34140.933} C_VEL
LIN {X 0,Y 752.659,Z 998.659,A -85,B 0,C 180,E1 34139.878,E2 34139.878} C_VEL
LIN {X 0,Y 752.523,Z 1022.288,A -85,B 0,C 180,E1 34138.489,E2 34138.489} C_VEL
LIN {X 0,Y 752.41,Z 1042.859,A -85,B 0,C 180,E1 34137.116,E2 34137.116} C_VEL
LIN {X 0,Y 752.344,Z 1061.291,A -85,B 0,C 180,E1 34135.758,E2 34135.758} C_VEL
LIN {X 0,Y 752.214,Z 1082.666,A -85,B 0,C 180,E1 34134,E2 34134} C_VEL
LIN {X 0,Y 752.157,Z 1098.985,A -85,B 0,C 180,E1 34132.495,E2 34132.495} C_VEL
LIN {X 0,Y 752.092,Z 1114.959,A -85,B 0,C 180,E1 34130.872,E2 34130.872} C_VEL
LIN {X 0,Y 752.02,Z 1131.872,A -85,B 0,C 180,E1 34128.929,E2 34128.929} C_VEL
LIN {X 0,Y 751.996,Z 1144.357,A -85,B 0,C 180,E1 34127.313,E2 34127.313} C_VEL
LIN {X 0,Y 751.96,Z 1155.265,A -85,B 0,C 180,E1 34125.738,E2 34125.738} C_VEL
LIN {X 0,Y 751.952,Z 1165.925,A -85,B 0,C 180,E1 34124.004,E2 34124.004} C_VEL
LIN {X 0,Y 751.91,Z 1177.004,A -85,B 0,C 180,E1 34121.894,E2 34121.894} C_VEL
LIN {X 0,Y 751.926,Z 1185.548,A -85,B 0,C 180,E1 34119.954,E2 34119.954} C_VEL
LIN {X 0,Y 751.919,Z 1193.115,A -85,B 0,C 180,E1 34117.794,E2 34117.794} C_VEL
LIN {X 0,Y 751.914,Z 1198.424,A -85,B 0,C 180,E1 34115.799,E2 34115.799} C_VEL
LIN {X 0,Y 751.909,Z 1202.282,A -85,B 0,C 180,E1 34113.735,E2 34113.735} C_VEL
LIN {X 0,Y 751.909,Z 1204.493,A -85,B 0,C 180,E1 34111.599,E2 34111.599} C_VEL
LIN {X 0,Y 751.89,Z 1204.874,A -85,B 0,C 180,E1 34109.542,E2 34109.542} C_VEL
LIN {X 0,Y 751.907,Z 1203.906,A -85,B 0,C 180,E1 34107.636,E2 34107.636} C_VEL
LIN {X 0,Y 751.907,Z 1201.051,A -85,B 0,C 180,E1 34105.499,E2 34105.499} C_VEL
LIN {X 0,Y 751.912,Z 1196.562,A -85,B 0,C 180,E1 34103.432,E2 34103.432} C_VEL
LIN {X 0,Y 751.92,Z 1190.624,A -85,B 0,C 180,E1 34101.434,E2 34101.434} C_VEL
LIN {X 0,Y 751.905,Z 1182.637,A -85,B 0,C 180,E1 34099.338,E2 34099.338} C_VEL
LIN {X 0,Y 751.935,Z 1173.109,A -85,B 0,C 180,E1 34097.325,E2 34097.325} C_VEL
LIN {X 0,Y 751.955,Z 1164.051,A -85,B 0,C 180,E1 34095.68,E2 34095.68} C_VEL
LIN {X 0,Y 751.954,Z 1154.207,A -85,B 0,C 180,E1 34094.101,E2 34094.101} C_VEL
LIN {X 0,Y 752.006,Z 1143.079,A -85,B 0,C 180,E1 34092.512,E2 34092.512} C_VEL
LIN {X 0,Y 752.063,Z 1128.618,A -85,B 0,C 180,E1 34090.667,E2 34090.667} C_VEL
LIN {X 0,Y 752.088,Z 1112.6,A -85,B 0,C 180,E1 34088.881,E2 34088.881} C_VEL
LIN {X 0,Y 752.166,Z 1097.962,A -85,B 0,C 180,E1 34087.406,E2 34087.406} C_VEL
LIN {X 0,Y 752.233,Z 1079.847,A -85,B 0,C 180,E1 34085.749,E2 34085.749} C_VEL
LIN {X 0,Y 752.348,Z 1059.77,A -85,B 0,C 180,E1 34084.126,E2 34084.126} C_VEL
LIN {X 0,Y 752.41,Z 1041.619,A -85,B 0,C 180,E1 34082.796,E2 34082.796} C_VEL
LIN {X 0,Y 752.554,Z 1019.504,A -85,B 0,C 180,E1 34081.337,E2 34081.337} C_VEL
LIN {X 0,Y 752.661,Z 997.818,A -85,B 0,C 180,E1 34080.076,E2 34080.076} C_VEL
LIN {X 0,Y 752.757,Z 978.507,A -85,B 0,C 180,E1 34079.065,E2 34079.065} C_VEL
LIN {X 0,Y 752.856,Z 958.67,A -85,B 0,C 180,E1 34078.134,E2 34078.134} C_VEL
LIN {X 0,Y 752.969,Z 934.985,A -85,B 0,C 180,E1 34077.148,E2 34077.148} C_VEL
LIN {X 0,Y 753.095,Z 909.057,A -85,B 0,C 180,E1 34076.24,E2 34076.24} C_VEL
LIN {X 0,Y 753.199,Z 884.115,A -85,B 0,C 180,E1 34075.503,E2 34075.503} C_VEL
LIN {X 0,Y 753.276,Z 856.426,A -85,B 0,C 180,E1 34074.856,E2 34074.856} C_VEL
LIN {X 0,Y 753.351,Z 829.765,A -85,B 0,C 180,E1 34074.393,E2 34074.393} C_VEL
LIN {X 0,Y 753.429,Z 761.411,A -85,B 0,C 180,E1 34073.583,E2 34073.583} C_VEL
LIN {X 0,Y 753.648,Z 538.106,A -85,B 0,C 180,E1 34070.959,E2 34070.959} C_VEL
LIN {X 0,Y 753.82,Z 344.439,A -85,B 0,C 180,E1 34068.594,E2 34068.594} C_VEL
LIN {X 0,Y 753.684,Z 314.597,A -85,B 0,C 180,E1 34068.011,E2 34068.011} C_VEL
LIN {X 0,Y 752.103,Z 311.339,A -85,B 0,C 180,E1 34067.839,E2 34067.839} C_VEL
LIN {X 0,Y 751.965,Z 310.567,A -85,B 0,C 180,E1 34067.802,E2 34067.802} C_VEL
LIN {X 0,Y 751.976,Z 310.561,A -85,B 0,C 180,E1 34064.808,E2 34064.808} C_VEL
LIN {X 0,Y 751.947,Z 310.566,A -85,B 0,C 180,E1 34061.87,E2 34061.87} C_VEL
LIN {X 0,Y 751.963,Z 310.566,A -85,B 0,C 180,E1 34059.054,E2 34059.054} C_VEL
LIN {X 0,Y 751.969,Z 310.562,A -85,B 0,C 180,E1 34056.279,E2 34056.279} C_VEL
LIN {X 0,Y 751.949,Z 310.566,A -85,B 0,C 180,E1 34053.493,E2 34053.493} C_VEL
LIN {X 0,Y 751.963,Z 310.56,A -85,B 0,C 180,E1 34050.616,E2 34050.616} C_VEL
LIN {X 0,Y 751.958,Z 310.565,A -85,B 0,C 180,E1 34047.65,E2 34047.65} C_VEL
LIN {X 0,Y 751.967,Z 310.56,A -85,B 0,C 180,E1 34044.846,E2 34044.846} C_VEL
LIN {X 0,Y 751.96,Z 310.565,A -85,B 0,C 180,E1 34041.941,E2 34041.941} C_VEL
LIN {X 0,Y 751.935,Z 310.566,A -85,B 0,C 180,E1 34039.094,E2 34039.094} C_VEL
LIN {X 0,Y 751.951,Z 310.564,A -85,B 0,C 180,E1 34036.294,E2 34036.294} C_VEL
LIN {X 0,Y 751.969,Z 310.565,A -85,B 0,C 180,E1 34033.378,E2 34033.378} C_VEL
LIN {X 0,Y 751.99,Z 310.74,A -85,B 0,C 180,E1 34030.711,E2 34030.711} C_VEL
LIN {X 0,Y 752.119,Z 372.388,A -85,B 0,C 180,E1 34028.602,E2 34028.602} C_VEL
LIN {X 0,Y 752.206,Z 439.764,A -85,B 0,C 180,E1 34026.219,E2 34026.219} C_VEL
LIN {X 0,Y 752.445,Z 480.212,A -85,B 0,C 180,E1 34024.726,E2 34024.726} C_VEL
LIN {X 0,Y 752.339,Z 553.11,A -85,B 0,C 180,E1 34021.938,E2 34021.938} C_VEL
LIN {X 0,Y 752.227,Z 630.122,A -85,B 0,C 180,E1 34019.048,E2 34019.048} C_VEL
LIN {X 0,Y 752.141,Z 707.526,A -85,B 0,C 180,E1 34016.189,E2 34016.189} C_VEL
LIN {X 0,Y 752.141,Z 711.123,A -85,B 0,C 180,E1 34016.057,E2 34016.057} C_VEL
LIN {X 0,Y 751.173,Z 718.163,A -85,B 0,C 180,E1 34015.818,E2 34015.818} C_VEL
LIN {X 0,Y 745.048,Z 737.088,A -85,B 0,C 180,E1 34015.244,E2 34015.244} C_VEL
LIN {X 0,Y 744.303,Z 743.131,A -85,B 0,C 180,E1 34015.036,E2 34015.036} C_VEL
LIN {X 0,Y 744.153,Z 822.626,A -85,B 0,C 180,E1 34012.123,E2 34012.123} C_VEL
LIN {X 0,Y 744.173,Z 836.783,A -85,B 0,C 180,E1 34011.628,E2 34011.628} C_VEL
LIN {X 0,Y 744.132,Z 951.59,A -85,B 0,C 180,E1 34010.506,E2 34010.506} C_VEL
LIN {X 0,Y 744.1,Z 966.389,A -85,B 0,C 180,E1 34010.231,E2 34010.231} C_VEL
LIN {X 0,Y 744.069,Z 980.37,A -85,B 0,C 180,E1 34009.822,E2 34009.822} C_VEL
LIN {X 0,Y 744.04,Z 993.035,A -85,B 0,C 180,E1 34009.312,E2 34009.312} C_VEL
LIN {X 0,Y 744.004,Z 1004.478,A -85,B 0,C 180,E1 34008.724,E2 34008.724} C_VEL
LIN {X 0,Y 743.98,Z 1016.493,A -85,B 0,C 180,E1 34007.937,E2 34007.937} C_VEL
LIN {X 0,Y 743.952,Z 1026.318,A -85,B 0,C 180,E1 34007.108,E2 34007.108} C_VEL
LIN {X 0,Y 743.939,Z 1033.894,A -85,B 0,C 180,E1 34006.317,E2 34006.317} C_VEL
LIN {X 0,Y 743.926,Z 1040.874,A -85,B 0,C 180,E1 34005.405,E2 34005.405} C_VEL
LIN {X 0,Y 743.92,Z 1047.482,A -85,B 0,C 180,E1 34004.246,E2 34004.246} C_VEL
LIN {X 0,Y 743.91,Z 1051.472,A -85,B 0,C 180,E1 34003.203,E2 34003.203} C_VEL
LIN {X 0,Y 743.919,Z 1053.797,A -85,B 0,C 180,E1 34002.235,E2 34002.235} C_VEL
LIN {X 0,Y 743.908,Z 1054.85,A -85,B 0,C 180,E1 34001.262,E2 34001.262} C_VEL
LIN {X 0,Y 743.917,Z 1054.528,A -85,B 0,C 180,E1 34000.12,E2 34000.12} C_VEL
LIN {X 0,Y 743.916,Z 1052.244,A -85,B 0,C 180,E1 33998.969,E2 33998.969} C_VEL
LIN {X 0,Y 743.918,Z 1049.056,A -85,B 0,C 180,E1 33998.036,E2 33998.036} C_VEL
LIN {X 0,Y 743.919,Z 1044.745,A -85,B 0,C 180,E1 33997.142,E2 33997.142} C_VEL
LIN {X 0,Y 743.926,Z 1038.866,A -85,B 0,C 180,E1 33996.22,E2 33996.22} C_VEL
LIN {X 0,Y 743.942,Z 1031.272,A -85,B 0,C 180,E1 33995.292,E2 33995.292} C_VEL
LIN {X 0,Y 743.967,Z 1021.313,A -85,B 0,C 180,E1 33994.357,E2 33994.357} C_VEL
LIN {X 0,Y 743.996,Z 1010.915,A -85,B 0,C 180,E1 33993.586,E2 33993.586} C_VEL
LIN {X 0,Y 744.006,Z 999.271,A -85,B 0,C 180,E1 33992.897,E2 33992.897} C_VEL
LIN {X 0,Y 744.064,Z 985.893,A -85,B 0,C 180,E1 33992.292,E2 33992.292} C_VEL
LIN {X 0,Y 744.083,Z 972.957,A -85,B 0,C 180,E1 33991.857,E2 33991.857} C_VEL
LIN {X 0,Y 744.12,Z 959.709,A -85,B 0,C 180,E1 33991.539,E2 33991.539} C_VEL
LIN {X 0,Y 744.134,Z 944.546,A -85,B 0,C 180,E1 33991.316,E2 33991.316} C_VEL
LIN {X 0,Y 744.131,Z 835.418,A -85,B 0,C 180,E1 33990.253,E2 33990.253} C_VEL
LIN {X 0,Y 744.28,Z 755.018,A -85,B 0,C 180,E1 33987.312,E2 33987.312} C_VEL
LIN {X 0,Y 744.449,Z 675.93,A -85,B 0,C 180,E1 33984.384,E2 33984.384} C_VEL
LIN {X 0,Y 744.653,Z 597.266,A -85,B 0,C 180,E1 33981.429,E2 33981.429} C_VEL
LIN {X 0,Y 744.86,Z 523.069,A -85,B 0,C 180,E1 33978.594,E2 33978.594} C_VEL
LIN {X 0,Y 744.866,Z 451.606,A -85,B 0,C 180,E1 33975.871,E2 33975.871} C_VEL
LIN {X 0,Y 744.831,Z 351.702,A -85,B 0,C 180,E1 33972.181,E2 33972.181} C_VEL
LIN {X 0,Y 744.898,Z 337.998,A -85,B 0,C 180,E1 33971.661,E2 33971.661} C_VEL
LIN {X 0,Y 746.183,Z 339.992,A -85,B 0,C 180,E1 33971.548,E2 33971.548} C_VEL
LIN {X 0,Y 747.78,Z 340.479,A -85,B 0,C 180,E1 33971.434,E2 33971.434} C_VEL
LIN {X 0,Y 747.316,Z 564.434,A -85,B 0,C 180,E1 33968.707,E2 33968.707} C_VEL
LIN {X 0,Y 746.823,Z 799.134,A -85,B 0,C 180,E1 33965.93,E2 33965.93} C_VEL
LIN {X 0,Y 746.69,Z 826.202,A -85,B 0,C 180,E1 33965.461,E2 33965.461} C_VEL
LIN {X 0,Y 746.51,Z 853.805,A -85,B 0,C 180,E1 33964.813,E2 33964.813} C_VEL
LIN {X 0,Y 746.314,Z 877.664,A -85,B 0,C 180,E1 33964.108,E2 33964.108} C_VEL
LIN {X 0,Y 746.121,Z 902.221,A -85,B 0,C 180,E1 33963.255,E2 33963.255} C_VEL
LIN {X 0,Y 745.826,Z 927.595,A -85,B 0,C 180,E1 33962.207,E2 33962.207} C_VEL
LIN {X 0,Y 745.626,Z 948.595,A -85,B 0,C 180,E1 33961.214,E2 33961.214} C_VEL
LIN {X 0,Y 745.429,Z 968.615,A -85,B 0,C 180,E1 33960.155,E2 33960.155} C_VEL
LIN {X 0,Y 745.176,Z 992.245,A -85,B 0,C 180,E1 33958.754,E2 33958.754} C_VEL
LIN {X 0,Y 744.938,Z 1013.704,A -85,B 0,C 180,E1 33957.306,E2 33957.306} C_VEL
LIN {X 0,Y 744.768,Z 1033.455,A -85,B 0,C 180,E1 33955.828,E2 33955.828} C_VEL
LIN {X 0,Y 744.532,Z 1053.548,A -85,B 0,C 180,E1 33954.139,E2 33954.139} C_VEL
LIN {X 0,Y 744.413,Z 1070.066,A -85,B 0,C 180,E1 33952.592,E2 33952.592} C_VEL
LIN {X 0,Y 744.288,Z 1087.627,A -85,B 0,C 180,E1 33950.768,E2 33950.768} C_VEL
LIN {X 0,Y 744.159,Z 1102.785,A -85,B 0,C 180,E1 33948.976,E2 33948.976} C_VEL
LIN {X 0,Y 744.089,Z 1114.559,A -85,B 0,C 180,E1 33947.429,E2 33947.429} C_VEL
LIN {X 0,Y 744.02,Z 1124.953,A -85,B 0,C 180,E1 33945.912,E2 33945.912} C_VEL
LIN {X 0,Y 744.005,Z 1134.769,A -85,B 0,C 180,E1 33944.309,E2 33944.309} C_VEL
LIN {X 0,Y 743.958,Z 1145.716,A -85,B 0,C 180,E1 33942.261,E2 33942.261} C_VEL
LIN {X 0,Y 743.939,Z 1155.362,A -85,B 0,C 180,E1 33940.064,E2 33940.064} C_VEL
LIN {X 0,Y 743.923,Z 1162.476,A -85,B 0,C 180,E1 33938.036,E2 33938.036} C_VEL
LIN {X 0,Y 743.916,Z 1167.978,A -85,B 0,C 180,E1 33936.019,E2 33936.019} C_VEL
LIN {X 0,Y 743.909,Z 1172.105,A -85,B 0,C 180,E1 33933.854,E2 33933.854} C_VEL
LIN {X 0,Y 743.906,Z 1174.345,A -85,B 0,C 180,E1 33931.772,E2 33931.772} C_VEL
LIN {X 0,Y 743.89,Z 1174.891,A -85,B 0,C 180,E1 33929.539,E2 33929.539} C_VEL
LIN {X 0,Y 743.906,Z 1173.955,A -85,B 0,C 180,E1 33927.613,E2 33927.613} C_VEL
LIN {X 0,Y 743.906,Z 1171.13,A -85,B 0,C 180,E1 33925.453,E2 33925.453} C_VEL
LIN {X 0,Y 743.915,Z 1166.872,A -85,B 0,C 180,E1 33923.441,E2 33923.441} C_VEL
LIN {X 0,Y 743.93,Z 1161.052,A -85,B 0,C 180,E1 33921.421,E2 33921.421} C_VEL
LIN {X 0,Y 743.917,Z 1153.04,A -85,B 0,C 180,E1 33919.276,E2 33919.276} C_VEL
LIN {X 0,Y 743.97,Z 1143.349,A -85,B 0,C 180,E1 33917.189,E2 33917.189} C_VEL
LIN {X 0,Y 744.001,Z 1134.324,A -85,B 0,C 180,E1 33915.525,E2 33915.525} C_VEL
LIN {X 0,Y 744.021,Z 1125.03,A -85,B 0,C 180,E1 33914.009,E2 33914.009} C_VEL
LIN {X 0,Y 744.092,Z 1114.576,A -85,B 0,C 180,E1 33912.483,E2 33912.483} C_VEL
LIN {X 0,Y 744.156,Z 1102.869,A -85,B 0,C 180,E1 33910.944,E2 33910.944} C_VEL
LIN {X 0,Y 744.272,Z 1088.379,A -85,B 0,C 180,E1 33909.228,E2 33909.228} C_VEL
LIN {X 0,Y 744.402,Z 1071.008,A -85,B 0,C 180,E1 33907.41,E2 33907.41} C_VEL
LIN {X 0,Y 744.526,Z 1055.031,A -85,B 0,C 180,E1 33905.905,E2 33905.905} C_VEL
LIN {X 0,Y 744.737,Z 1035.922,A -85,B 0,C 180,E1 33904.276,E2 33904.276} C_VEL
LIN {X 0,Y 744.929,Z 1014.986,A -85,B 0,C 180,E1 33902.696,E2 33902.696} C_VEL
LIN {X 0,Y 745.121,Z 995.307,A -85,B 0,C 180,E1 33901.356,E2 33901.356} C_VEL
LIN {X 0,Y 745.417,Z 970.28,A -85,B 0,C 180,E1 33899.846,E2 33899.846} C_VEL
LIN {X 0,Y 745.623,Z 949.443,A -85,B 0,C 180,E1 33898.738,E2 33898.738} C_VEL
LIN {X 0,Y 745.821,Z 928.719,A -85,B 0,C 180,E1 33897.754,E2 33897.754} C_VEL
LIN {X 0,Y 746.099,Z 903.898,A -85,B 0,C 180,E1 33896.717,E2 33896.717} C_VEL
LIN {X 0,Y 746.312,Z 878.495,A -85,B 0,C 180,E1 33895.828,E2 33895.828} C_VEL
LIN {X 0,Y 746.5,Z 854.385,A -85,B 0,C 180,E1 33895.112,E2 33895.112} C_VEL
LIN {X 0,Y 746.686,Z 826.711,A -85,B 0,C 180,E1 33894.46,E2 33894.46} C_VEL
LIN {X 0,Y 746.822,Z 799.682,A -85,B 0,C 180,E1 33893.988,E2 33893.988} C_VEL
LIN {X 0,Y 747.013,Z 718.15,A -85,B 0,C 180,E1 33893.018,E2 33893.018} C_VEL
LIN {X 0,Y 747.43,Z 498.869,A -85,B 0,C 180,E1 33890.414,E2 33890.414} C_VEL
LIN {X 0,Y 747.742,Z 325.323,A -85,B 0,C 180,E1 33888.283,E2 33888.283} C_VEL
LIN {X 0,Y 746.555,Z 320.745,A -85,B 0,C 180,E1 33888.131,E2 33888.131} C_VEL
LIN {X 0,Y 746.408,Z 317.76,A -85,B 0,C 180,E1 33887.914,E2 33887.914} C_VEL
LIN {X 0,Y 744.028,Z 311.556,A -85,B 0,C 180,E1 33887.289,E2 33887.289} C_VEL
LIN {X 0,Y 744.004,Z 311.555,A -85,B 0,C 180,E1 33884.55,E2 33884.55} C_VEL
LIN {X 0,Y 744.041,Z 311.554,A -85,B 0,C 180,E1 33881.596,E2 33881.596} C_VEL
LIN {X 0,Y 744.007,Z 311.556,A -85,B 0,C 180,E1 33878.776,E2 33878.776} C_VEL
LIN {X 0,Y 744.012,Z 311.555,A -85,B 0,C 180,E1 33875.965,E2 33875.965} C_VEL
LIN {X 0,Y 744.023,Z 311.551,A -85,B 0,C 180,E1 33873.153,E2 33873.153} C_VEL
LIN {X 0,Y 744.004,Z 311.554,A -85,B 0,C 180,E1 33870.353,E2 33870.353} C_VEL
LIN {X 0,Y 744.037,Z 311.555,A -85,B 0,C 180,E1 33867.448,E2 33867.448} C_VEL
LIN {X 0,Y 744.003,Z 311.55,A -85,B 0,C 180,E1 33864.521,E2 33864.521} C_VEL
LIN {X 0,Y 744.03,Z 311.555,A -85,B 0,C 180,E1 33861.689,E2 33861.689} C_VEL
LIN {X 0,Y 744.025,Z 311.552,A -85,B 0,C 180,E1 33858.816,E2 33858.816} C_VEL
LIN {X 0,Y 744.021,Z 311.552,A -85,B 0,C 180,E1 33855.912,E2 33855.912} C_VEL
LIN {X 0,Y 744.036,Z 311.552,A -85,B 0,C 180,E1 33853.024,E2 33853.024} C_VEL
LIN {X 0,Y 744.031,Z 311.55,A -85,B 0,C 180,E1 33849.983,E2 33849.983} C_VEL
LIN {X 0,Y 744.023,Z 311.55,A -85,B 0,C 180,E1 33847.102,E2 33847.102} C_VEL
LIN {X 0,Y 744.035,Z 311.554,A -85,B 0,C 180,E1 33844.084,E2 33844.084} C_VEL
LIN {X 0,Y 744.006,Z 311.551,A -85,B 0,C 180,E1 33841.232,E2 33841.232} C_VEL
LIN {X 0,Y 744.04,Z 311.553,A -85,B 0,C 180,E1 33838.306,E2 33838.306} C_VEL
LIN {X 0,Y 744.009,Z 311.556,A -85,B 0,C 180,E1 33835.452,E2 33835.452} C_VEL
LIN {X 0,Y 744.013,Z 311.549,A -85,B 0,C 180,E1 33832.587,E2 33832.587} C_VEL
LIN {X 0,Y 744.022,Z 311.55,A -85,B 0,C 180,E1 33829.782,E2 33829.782} C_VEL
LIN {X 0,Y 744.004,Z 311.555,A -85,B 0,C 180,E1 33826.987,E2 33826.987} C_VEL
LIN {X 0,Y 744.037,Z 311.553,A -85,B 0,C 180,E1 33824.089,E2 33824.089} C_VEL
LIN {X 0,Y 744.003,Z 311.554,A -85,B 0,C 180,E1 33821.183,E2 33821.183} C_VEL
LIN {X 0,Y 744.023,Z 311.542,A -85,B 0,C 180,E1 33818.394,E2 33818.394} C_VEL
LIN {X 0,Y 744.058,Z 311.691,A -85,B 0,C 180,E1 33818.042,E2 33818.042} C_VEL
LIN {X 0,Y 745.484,Z 315.257,A -85,B 0,C 180,E1 33817.609,E2 33817.609} C_VEL
LIN {X 0,Y 746.492,Z 316.692,A -85,B 0,C 180,E1 33817.392,E2 33817.392} C_VEL
LIN {X 0,Y 748.113,Z 320.301,A -85,B 0,C 180,E1 33816.945,E2 33816.945} C_VEL
LIN {X 0,Y 747.809,Z 354.324,A -85,B 0,C 180,E1 33814.413,E2 33814.413} C_VEL
LIN {X 0,Y 747.456,Z 391.086,A -85,B 0,C 180,E1 33811.822,E2 33811.822} C_VEL
LIN {X 0,Y 747.125,Z 428.637,A -85,B 0,C 180,E1 33809.298,E2 33809.298} C_VEL
LIN {X 0,Y 746.813,Z 468.207,A -85,B 0,C 180,E1 33806.751,E2 33806.751} C_VEL
LIN {X 0,Y 746.494,Z 510.64,A -85,B 0,C 180,E1 33804.129,E2 33804.129} C_VEL
LIN {X 0,Y 747.026,Z 522.962,A -85,B 0,C 180,E1 33803.347,E2 33803.347} C_VEL
LIN {X 0,Y 748.749,Z 530.652,A -85,B 0,C 180,E1 33802.775,E2 33802.775} C_VEL
LIN {X 0,Y 750.502,Z 534.787,A -85,B 0,C 180,E1 33802.312,E2 33802.312} C_VEL
LIN {X 0,Y 751.849,Z 536.691,A -85,B 0,C 180,E1 33801.897,E2 33801.897} C_VEL
LIN {X 0,Y 752.83,Z 537.128,A -85,B 0,C 180,E1 33801.469,E2 33801.469} C_VEL
LIN {X 0,Y 753.271,Z 535.875,A -85,B 0,C 180,E1 33801.01,E2 33801.01} C_VEL
LIN {X 0,Y 752.965,Z 532.967,A -85,B 0,C 180,E1 33800.609,E2 33800.609} C_VEL
LIN {X 0,Y 751.976,Z 528.489,A -85,B 0,C 180,E1 33800.282,E2 33800.282} C_VEL
LIN {X 0,Y 750.474,Z 522.578,A -85,B 0,C 180,E1 33800.054,E2 33800.054} C_VEL
LIN {X 0,Y 748.608,Z 513.939,A -85,B 0,C 180,E1 33799.92,E2 33799.92} C_VEL
LIN {X 0,Y 747.64,Z 501.89,A -85,B 0,C 180,E1 33799.857,E2 33799.857} C_VEL
LIN {X 0,Y 747.461,Z 317.212,A -85,B 0,C 180,E1 33799.846,E2 33799.846} C_VEL
LIN {X 0,Y 744.98,Z 314.478,A -85,B 0,C 180,E1 33799.684,E2 33799.684} C_VEL
LIN {X 0,Y 744.022,Z 311.553,A -85,B 0,C 180,E1 33799.607,E2 33799.607} C_VEL
LIN {X 0,Y 744.009,Z 311.555,A -85,B 0,C 180,E1 33796.627,E2 33796.627} C_VEL
LIN {X 0,Y 744.023,Z 311.631,A -85,B 0,C 180,E1 33794.58,E2 33794.58} C_VEL
LIN {X 0,Y 745.346,Z 315.116,A -85,B 0,C 180,E1 33794.244,E2 33794.244} C_VEL
LIN {X 0,Y 746.924,Z 318.816,A -85,B 0,C 180,E1 33793.878,E2 33793.878} C_VEL
LIN {X 0,Y 746.794,Z 351.111,A -85,B 0,C 180,E1 33791.79,E2 33791.79} C_VEL
LIN {X 0,Y 747.807,Z 355.704,A -85,B 0,C 180,E1 33791.662,E2 33791.662} C_VEL
LIN {X 0,Y 747.359,Z 570.243,A -85,B 0,C 180,E1 33789.042,E2 33789.042} C_VEL
LIN {X 0,Y 746.927,Z 795.075,A -85,B 0,C 180,E1 33786.391,E2 33786.391} C_VEL
LIN {X 0,Y 746.816,Z 833.09,A -85,B 0,C 180,E1 33785.917,E2 33785.917} C_VEL
LIN {X 0,Y 746.66,Z 859.063,A -85,B 0,C 180,E1 33785.445,E2 33785.445} C_VEL
LIN {X 0,Y 746.488,Z 885.778,A -85,B 0,C 180,E1 33784.806,E2 33784.806} C_VEL
LIN {X 0,Y 746.282,Z 913.631,A -85,B 0,C 180,E1 33783.965,E2 33783.965} C_VEL
LIN {X 0,Y 746.009,Z 939.521,A -85,B 0,C 180,E1 33783.012,E2 33783.012} C_VEL
LIN {X 0,Y 745.814,Z 959.719,A -85,B 0,C 180,E1 33782.156,E2 33782.156} C_VEL
LIN {X 0,Y 745.614,Z 980.34,A -85,B 0,C 180,E1 33781.172,E2 33781.172} C_VEL
LIN {X 0,Y 745.389,Z 1003.457,A -85,B 0,C 180,E1 33779.933,E2 33779.933} C_VEL
LIN {X 0,Y 745.113,Z 1026.267,A -85,B 0,C 180,E1 33778.535,E2 33778.535} C_VEL
LIN {X 0,Y 744.924,Z 1045.284,A -85,B 0,C 180,E1 33777.238,E2 33777.238} C_VEL
LIN {X 0,Y 744.733,Z 1066.222,A -85,B 0,C 180,E1 33775.656,E2 33775.656} C_VEL
LIN {X 0,Y 744.531,Z 1085.464,A -85,B 0,C 180,E1 33774.01,E2 33774.01} C_VEL
LIN {X 0,Y 744.392,Z 1102.253,A -85,B 0,C 180,E1 33772.424,E2 33772.424} C_VEL
LIN {X 0,Y 744.248,Z 1120.125,A -85,B 0,C 180,E1 33770.526,E2 33770.526} C_VEL
LIN {X 0,Y 744.144,Z 1133.571,A -85,B 0,C 180,E1 33768.923,E2 33768.923} C_VEL
LIN {X 0,Y 744.087,Z 1145.426,A -85,B 0,C 180,E1 33767.355,E2 33767.355} C_VEL
LIN {X 0,Y 744.032,Z 1157.358,A -85,B 0,C 180,E1 33765.59,E2 33765.59} C_VEL
LIN {X 0,Y 743.978,Z 1169.839,A -85,B 0,C 180,E1 33763.444,E2 33763.444} C_VEL
LIN {X 0,Y 743.93,Z 1178.437,A -85,B 0,C 180,E1 33761.709,E2 33761.709} C_VEL
LIN {X 0,Y 743.931,Z 1186.279,A -85,B 0,C 180,E1 33759.869,E2 33759.869} C_VEL
LIN {X 0,Y 743.92,Z 1193.594,A -85,B 0,C 180,E1 33757.723,E2 33757.723} C_VEL
LIN {X 0,Y 743.916,Z 1199.111,A -85,B 0,C 180,E1 33755.552,E2 33755.552} C_VEL
LIN {X 0,Y 743.915,Z 1202.588,A -85,B 0,C 180,E1 33753.544,E2 33753.544} C_VEL
LIN {X 0,Y 743.913,Z 1204.585,A -85,B 0,C 180,E1 33751.462,E2 33751.462} C_VEL
LIN {X 0,Y 743.889,Z 1204.853,A -85,B 0,C 180,E1 33749.46,E2 33749.46} C_VEL
LIN {X 0,Y 743.906,Z 1203.906,A -85,B 0,C 180,E1 33747.611,E2 33747.611} C_VEL
LIN {X 0,Y 743.908,Z 1201.175,A -85,B 0,C 180,E1 33745.528,E2 33745.528} C_VEL
LIN {X 0,Y 743.918,Z 1196.952,A -85,B 0,C 180,E1 33743.516,E2 33743.516} C_VEL
LIN {X 0,Y 743.926,Z 1190.892,A -85,B 0,C 180,E1 33741.419,E2 33741.419} C_VEL
LIN {X 0,Y 743.918,Z 1182.855,A -85,B 0,C 180,E1 33739.275,E2 33739.275} C_VEL
LIN {X 0,Y 743.97,Z 1173.112,A -85,B 0,C 180,E1 33737.187,E2 33737.187} C_VEL
LIN {X 0,Y 743.999,Z 1164.054,A -85,B 0,C 180,E1 33735.523,E2 33735.523} C_VEL
LIN {X 0,Y 744.023,Z 1154.183,A -85,B 0,C 180,E1 33733.923,E2 33733.923} C_VEL
LIN {X 0,Y 744.103,Z 1143.026,A -85,B 0,C 180,E1 33732.312,E2 33732.312} C_VEL
LIN {X 0,Y 744.222,Z 1127.813,A -85,B 0,C 180,E1 33730.36,E2 33730.36} C_VEL
LIN {X 0,Y 744.304,Z 1112.011,A -85,B 0,C 180,E1 33728.587,E2 33728.587} C_VEL
LIN {X 0,Y 744.426,Z 1097.11,A -85,B 0,C 180,E1 33727.075,E2 33727.075} C_VEL
LIN {X 0,Y 744.626,Z 1077.879,A -85,B 0,C 180,E1 33725.315,E2 33725.315} C_VEL
LIN {X 0,Y 744.783,Z 1059.054,A -85,B 0,C 180,E1 33723.788,E2 33723.788} C_VEL
LIN {X 0,Y 744.981,Z 1039.206,A -85,B 0,C 180,E1 33722.329,E2 33722.329} C_VEL
LIN {X 0,Y 745.246,Z 1015.868,A -85,B 0,C 180,E1 33720.81,E2 33720.81} C_VEL
LIN {X 0,Y 745.442,Z 996.219,A -85,B 0,C 180,E1 33719.667,E2 33719.667} C_VEL
LIN {X 0,Y 745.645,Z 974.955,A -85,B 0,C 180,E1 33718.557,E2 33718.557} C_VEL
LIN {X 0,Y 745.965,Z 948.409,A -85,B 0,C 180,E1 33717.349,E2 33717.349} C_VEL
LIN {X 0,Y 746.165,Z 925.624,A -85,B 0,C 180,E1 33716.461,E2 33716.461} C_VEL
LIN {X 0,Y 746.335,Z 904.676,A -85,B 0,C 180,E1 33715.753,E2 33715.753} C_VEL
LIN {X 0,Y 746.523,Z 881.473,A -85,B 0,C 180,E1 33715.081,E2 33715.081} C_VEL
LIN {X 0,Y 746.703,Z 854.868,A -85,B 0,C 180,E1 33714.467,E2 33714.467} C_VEL
LIN {X 0,Y 746.829,Z 827.221,A -85,B 0,C 180,E1 33713.996,E2 33713.996} C_VEL
LIN {X 0,Y 747.319,Z 588.059,A -85,B 0,C 180,E1 33711.171,E2 33711.171} C_VEL
LIN {X 0,Y 747.74,Z 381.474,A -85,B 0,C 180,E1 33708.657,E2 33708.657} C_VEL
LIN {X 0,Y 747.764,Z 343.777,A -85,B 0,C 180,E1 33708.17,E2 33708.17} C_VEL
LIN {X 0,Y 747.65,Z 318.344,A -85,B 0,C 180,E1 33707.667,E2 33707.667} C_VEL
LIN {X 0,Y 746.409,Z 316.341,A -85,B 0,C 180,E1 33707.541,E2 33707.541} C_VEL
LIN {X 0,Y 744.423,Z 313.295,A -85,B 0,C 180,E1 33707.34,E2 33707.34} C_VEL
LIN {X 0,Y 744.007,Z 311.555,A -85,B 0,C 180,E1 33707.259,E2 33707.259} C_VEL
LIN {X 0,Y 744.031,Z 311.553,A -85,B 0,C 180,E1 33704.333,E2 33704.333} C_VEL
LIN {X 0,Y 744.035,Z 311.552,A -85,B 0,C 180,E1 33701.419,E2 33701.419} C_VEL
LIN {X 0,Y 744.029,Z 311.552,A -85,B 0,C 180,E1 33698.419,E2 33698.419} C_VEL
LIN {X 0,Y 743.999,Z 311.551,A -85,B 0,C 180,E1 33695.492,E2 33695.492} C_VEL
LIN {X 0,Y 744.016,Z 311.555,A -85,B 0,C 180,E1 33692.701,E2 33692.701} C_VEL
LIN {X 0,Y 744.029,Z 311.554,A -85,B 0,C 180,E1 33689.818,E2 33689.818} C_VEL
LIN {X 0,Y 744.012,Z 311.551,A -85,B 0,C 180,E1 33686.998,E2 33686.998} C_VEL
LIN {X 0,Y 744.03,Z 311.548,A -85,B 0,C 180,E1 33683.945,E2 33683.945} C_VEL
LIN {X 0,Y 744.026,Z 311.555,A -85,B 0,C 180,E1 33681.028,E2 33681.028} C_VEL
LIN {X 0,Y 744.038,Z 311.551,A -85,B 0,C 180,E1 33678.085,E2 33678.085} C_VEL
LIN {X 0,Y 743.995,Z 311.555,A -85,B 0,C 180,E1 33675.113,E2 33675.113} C_VEL
LIN {X 0,Y 743.996,Z 311.556,A -85,B 0,C 180,E1 33672.417,E2 33672.417} C_VEL
LIN {X 0,Y 744.029,Z 311.67,A -85,B 0,C 180,E1 33670.845,E2 33670.845} C_VEL
LIN {X 0,Y 744.33,Z 317.228,A -85,B 0,C 180,E1 33670.65,E2 33670.65} C_VEL
LIN {X 0,Y 744.348,Z 394.432,A -85,B 0,C 180,E1 33667.992,E2 33667.992} C_VEL
LIN {X 0,Y 744.824,Z 486.284,A -85,B 0,C 180,E1 33664.697,E2 33664.697} C_VEL
LIN {X 0,Y 744.823,Z 534.246,A -85,B 0,C 180,E1 33662.886,E2 33662.886} C_VEL
LIN {X 0,Y 744.62,Z 607.94,A -85,B 0,C 180,E1 33660.077,E2 33660.077} C_VEL
LIN {X 0,Y 744.425,Z 687.021,A -85,B 0,C 180,E1 33657.113,E2 33657.113} C_VEL
LIN {X 0,Y 744.303,Z 743.131,A -85,B 0,C 180,E1 33655.036,E2 33655.036} C_VEL
LIN {X 0,Y 743.32,Z 750.169,A -85,B 0,C 180,E1 33654.795,E2 33654.795} C_VEL
LIN {X 0,Y 737.164,Z 769.062,A -85,B 0,C 180,E1 33654.21,E2 33654.21} C_VEL
LIN {X 0,Y 736.412,Z 775.104,A -85,B 0,C 180,E1 33654,E2 33654} C_VEL
LIN {X 0,Y 736.288,Z 836.734,A -85,B 0,C 180,E1 33651.744,E2 33651.744} C_VEL
LIN {X 0,Y 736.241,Z 951.7,A -85,B 0,C 180,E1 33650.608,E2 33650.608} C_VEL
LIN {X 0,Y 736.196,Z 966.658,A -85,B 0,C 180,E1 33650.324,E2 33650.324} C_VEL
LIN {X 0,Y 736.149,Z 980.632,A -85,B 0,C 180,E1 33649.909,E2 33649.909} C_VEL
LIN {X 0,Y 736.107,Z 993.258,A -85,B 0,C 180,E1 33649.394,E2 33649.394} C_VEL
LIN {X 0,Y 736.054,Z 1005.439,A -85,B 0,C 180,E1 33648.754,E2 33648.754} C_VEL
LIN {X 0,Y 736.006,Z 1017.648,A -85,B 0,C 180,E1 33647.924,E2 33647.924} C_VEL
LIN {X 0,Y 735.97,Z 1027.669,A -85,B 0,C 180,E1 33647.046,E2 33647.046} C_VEL
LIN {X 0,Y 735.949,Z 1035.674,A -85,B 0,C 180,E1 33646.165,E2 33646.165} C_VEL
LIN {X 0,Y 735.924,Z 1043.481,A -85,B 0,C 180,E1 33645.04,E2 33645.04} C_VEL
LIN {X 0,Y 735.921,Z 1048.373,A -85,B 0,C 180,E1 33644.07,E2 33644.07} C_VEL
LIN {X 0,Y 735.913,Z 1051.86,A -85,B 0,C 180,E1 33643.096,E2 33643.096} C_VEL
LIN {X 0,Y 735.919,Z 1054.024,A -85,B 0,C 180,E1 33642.117,E2 33642.117} C_VEL
LIN {X 0,Y 735.913,Z 1054.999,A -85,B 0,C 180,E1 33640.968,E2 33640.968} C_VEL
LIN {X 0,Y 735.917,Z 1054.055,A -85,B 0,C 180,E1 33639.811,E2 33639.811} C_VEL
LIN {X 0,Y 735.915,Z 1051.855,A -85,B 0,C 180,E1 33638.813,E2 33638.813} C_VEL
LIN {X 0,Y 735.921,Z 1048.591,A -85,B 0,C 180,E1 33637.892,E2 33637.892} C_VEL
LIN {X 0,Y 735.923,Z 1043.532,A -85,B 0,C 180,E1 33636.88,E2 33636.88} C_VEL
LIN {X 0,Y 735.949,Z 1035.921,A -85,B 0,C 180,E1 33635.776,E2 33635.776} C_VEL
LIN {X 0,Y 735.973,Z 1027.801,A -85,B 0,C 180,E1 33634.877,E2 33634.877} C_VEL
LIN {X 0,Y 736.006,Z 1017.47,A -85,B 0,C 180,E1 33633.972,E2 33633.972} C_VEL
LIN {X 0,Y 736.053,Z 1005.376,A -85,B 0,C 180,E1 33633.152,E2 33633.152} C_VEL
LIN {X 0,Y 736.104,Z 992.779,A -85,B 0,C 180,E1 33632.494,E2 33632.494} C_VEL
LIN {X 0,Y 736.146,Z 979.663,A -85,B 0,C 180,E1 33631.968,E2 33631.968} C_VEL
LIN {X 0,Y 736.213,Z 964.326,A -85,B 0,C 180,E1 33631.532,E2 33631.532} C_VEL
LIN {X 0,Y 736.242,Z 950.002,A -85,B 0,C 180,E1 33631.279,E2 33631.279} C_VEL
LIN {X 0,Y 736.248,Z 835.738,A -85,B 0,C 180,E1 33630.149,E2 33630.149} C_VEL
LIN {X 0,Y 736.469,Z 754.712,A -85,B 0,C 180,E1 33627.153,E2 33627.153} C_VEL
LIN {X 0,Y 736.729,Z 675.787,A -85,B 0,C 180,E1 33624.2,E2 33624.2} C_VEL
LIN {X 0,Y 737.033,Z 597.094,A -85,B 0,C 180,E1 33621.213,E2 33621.213} C_VEL
LIN {X 0,Y 737.22,Z 531.648,A -85,B 0,C 180,E1 33618.711,E2 33618.711} C_VEL
LIN {X 0,Y 737.308,Z 458.658,A -85,B 0,C 180,E1 33615.917,E2 33615.917} C_VEL
LIN {X 0,Y 737.297,Z 353.917,A -85,B 0,C 180,E1 33612.031,E2 33612.031} C_VEL
LIN {X 0,Y 737.369,Z 353.215,A -85,B 0,C 180,E1 33611.989,E2 33611.989} C_VEL
LIN {X 0,Y 738.603,Z 355.161,A -85,B 0,C 180,E1 33611.878,E2 33611.878} C_VEL
LIN {X 0,Y 740.442,Z 355.444,A -85,B 0,C 180,E1 33611.747,E2 33611.747} C_VEL
LIN {X 0,Y 741.729,Z 355.059,A -85,B 0,C 180,E1 33611.663,E2 33611.663} C_VEL
LIN {X 0,Y 741.03,Z 575.675,A -85,B 0,C 180,E1 33608.961,E2 33608.961} C_VEL
LIN {X 0,Y 740.325,Z 799.172,A -85,B 0,C 180,E1 33606.296,E2 33606.296} C_VEL
LIN {X 0,Y 740.128,Z 826.27,A -85,B 0,C 180,E1 33605.823,E2 33605.823} C_VEL
LIN {X 0,Y 739.852,Z 853.619,A -85,B 0,C 180,E1 33605.178,E2 33605.178} C_VEL
LIN {X 0,Y 739.565,Z 877.07,A -85,B 0,C 180,E1 33604.483,E2 33604.483} C_VEL
LIN {X 0,Y 739.288,Z 900.206,A -85,B 0,C 180,E1 33603.679,E2 33603.679} C_VEL
LIN {X 0,Y 738.839,Z 926.72,A -85,B 0,C 180,E1 33602.591,E2 33602.591} C_VEL
LIN {X 0,Y 738.518,Z 948.524,A -85,B 0,C 180,E1 33601.554,E2 33601.554} C_VEL
LIN {X 0,Y 738.212,Z 969.434,A -85,B 0,C 180,E1 33600.436,E2 33600.436} C_VEL
LIN {X 0,Y 737.795,Z 994.246,A -85,B 0,C 180,E1 33598.936,E2 33598.936} C_VEL
LIN {X 0,Y 737.463,Z 1015.183,A -85,B 0,C 180,E1 33597.5,E2 33597.5} C_VEL
LIN {X 0,Y 737.177,Z 1036.153,A -85,B 0,C 180,E1 33595.898,E2 33595.898} C_VEL
LIN {X 0,Y 736.853,Z 1054.955,A -85,B 0,C 180,E1 33594.279,E2 33594.279} C_VEL
LIN {X 0,Y 736.68,Z 1070.928,A -85,B 0,C 180,E1 33592.758,E2 33592.758} C_VEL
LIN {X 0,Y 736.461,Z 1089.012,A -85,B 0,C 180,E1 33590.838,E2 33590.838} C_VEL
LIN {X 0,Y 736.296,Z 1102.79,A -85,B 0,C 180,E1 33589.187,E2 33589.187} C_VEL
LIN {X 0,Y 736.189,Z 1114.499,A -85,B 0,C 180,E1 33587.631,E2 33587.631} C_VEL
LIN {X 0,Y 736.088,Z 1124.957,A -85,B 0,C 180,E1 33586.089,E2 33586.089} C_VEL
LIN {X 0,Y 736.048,Z 1134.72,A -85,B 0,C 180,E1 33584.476,E2 33584.476} C_VEL
LIN {X 0,Y 735.997,Z 1145.332,A -85,B 0,C 180,E1 33582.476,E2 33582.476} C_VEL
LIN {X 0,Y 735.951,Z 1155.362,A -85,B 0,C 180,E1 33580.174,E2 33580.174} C_VEL
LIN {X 0,Y 735.929,Z 1162.476,A -85,B 0,C 180,E1 33578.124,E2 33578.124} C_VEL
LIN {X 0,Y 735.92,Z 1167.98,A -85,B 0,C 180,E1 33576.084,E2 33576.084} C_VEL
LIN {X 0,Y 735.91,Z 1172.107,A -85,B 0,C 180,E1 33573.896,E2 33573.896} C_VEL
LIN {X 0,Y 735.907,Z 1174.345,A -85,B 0,C 180,E1 33571.792,E2 33571.792} C_VEL
LIN {X 0,Y 735.89,Z 1174.894,A -85,B 0,C 180,E1 33569.534,E2 33569.534} C_VEL
LIN {X 0,Y 735.905,Z 1173.955,A -85,B 0,C 180,E1 33567.587,E2 33567.587} C_VEL
LIN {X 0,Y 735.906,Z 1171.13,A -85,B 0,C 180,E1 33565.403,E2 33565.403} C_VEL
LIN {X 0,Y 735.914,Z 1166.869,A -85,B 0,C 180,E1 33563.369,E2 33563.369} C_VEL
LIN {X 0,Y 735.933,Z 1161.047,A -85,B 0,C 180,E1 33561.327,E2 33561.327} C_VEL
LIN {X 0,Y 735.931,Z 1153.185,A -85,B 0,C 180,E1 33559.194,E2 33559.194} C_VEL
LIN {X 0,Y 735.99,Z 1143.348,A -85,B 0,C 180,E1 33557.048,E2 33557.048} C_VEL
LIN {X 0,Y 736.039,Z 1134.321,A -85,B 0,C 180,E1 33555.365,E2 33555.365} C_VEL
LIN {X 0,Y 736.092,Z 1124.928,A -85,B 0,C 180,E1 33553.817,E2 33553.817} C_VEL
LIN {X 0,Y 736.187,Z 1114.573,A -85,B 0,C 180,E1 33552.289,E2 33552.289} C_VEL
LIN {X 0,Y 736.293,Z 1102.865,A -85,B 0,C 180,E1 33550.733,E2 33550.733} C_VEL
LIN {X 0,Y 736.461,Z 1088.374,A -85,B 0,C 180,E1 33548.997,E2 33548.997} C_VEL
LIN {X 0,Y 736.675,Z 1071.006,A -85,B 0,C 180,E1 33547.16,E2 33547.16} C_VEL
LIN {X 0,Y 736.855,Z 1054.38,A -85,B 0,C 180,E1 33545.579,E2 33545.579} C_VEL
LIN {X 0,Y 737.212,Z 1034.535,A -85,B 0,C 180,E1 33543.881,E2 33543.881} C_VEL
LIN {X 0,Y 737.471,Z 1014.035,A -85,B 0,C 180,E1 33542.327,E2 33542.327} C_VEL
LIN {X 0,Y 737.855,Z 992.309,A -85,B 0,C 180,E1 33540.847,E2 33540.847} C_VEL
LIN {X 0,Y 738.216,Z 968.669,A -85,B 0,C 180,E1 33539.431,E2 33539.431} C_VEL
LIN {X 0,Y 738.517,Z 948.636,A -85,B 0,C 180,E1 33538.362,E2 33538.362} C_VEL
LIN {X 0,Y 738.842,Z 926.724,A -85,B 0,C 180,E1 33537.32,E2 33537.32} C_VEL
LIN {X 0,Y 739.288,Z 900.182,A -85,B 0,C 180,E1 33536.23,E2 33536.23} C_VEL
LIN {X 0,Y 739.563,Z 877.748,A -85,B 0,C 180,E1 33535.449,E2 33535.449} C_VEL
LIN {X 0,Y 739.844,Z 854.102,A -85,B 0,C 180,E1 33534.745,E2 33534.745} C_VEL
LIN {X 0,Y 740.127,Z 826.685,A -85,B 0,C 180,E1 33534.096,E2 33534.096} C_VEL
LIN {X 0,Y 740.323,Z 799.64,A -85,B 0,C 180,E1 33533.621,E2 33533.621} C_VEL
LIN {X 0,Y 740.659,Z 700.173,A -85,B 0,C 180,E1 33532.432,E2 33532.432} C_VEL
LIN {X 0,Y 741.29,Z 485.826,A -85,B 0,C 180,E1 33529.859,E2 33529.859} C_VEL
LIN {X 0,Y 741.699,Z 327.345,A -85,B 0,C 180,E1 33527.892,E2 33527.892} C_VEL
LIN {X 0,Y 739.893,Z 321.718,A -85,B 0,C 180,E1 33527.694,E2 33527.694} C_VEL
LIN {X 0,Y 738.918,Z 319.593,A -85,B 0,C 180,E1 33527.518,E2 33527.518} C_VEL
LIN {X 0,Y 736.113,Z 312.872,A -85,B 0,C 180,E1 33526.839,E2 33526.839} C_VEL
LIN {X 0,Y 736.065,Z 312.546,A -85,B 0,C 180,E1 33526.729,E2 33526.729} C_VEL
LIN {X 0,Y 736.099,Z 312.544,A -85,B 0,C 180,E1 33523.841,E2 33523.841} C_VEL
LIN {X 0,Y 736.065,Z 312.545,A -85,B 0,C 180,E1 33520.902,E2 33520.902} C_VEL
LIN {X 0,Y 736.093,Z 312.545,A -85,B 0,C 180,E1 33518.076,E2 33518.076} C_VEL
LIN {X 0,Y 736.078,Z 312.543,A -85,B 0,C 180,E1 33515.142,E2 33515.142} C_VEL
LIN {X 0,Y 736.092,Z 312.541,A -85,B 0,C 180,E1 33512.195,E2 33512.195} C_VEL
LIN {X 0,Y 736.101,Z 312.531,A -85,B 0,C 180,E1 33509.276,E2 33509.276} C_VEL
LIN {X 0,Y 736.095,Z 312.543,A -85,B 0,C 180,E1 33506.285,E2 33506.285} C_VEL
LIN {X 0,Y 736.093,Z 312.54,A -85,B 0,C 180,E1 33503.284,E2 33503.284} C_VEL
LIN {X 0,Y 736.092,Z 312.536,A -85,B 0,C 180,E1 33500.35,E2 33500.35} C_VEL
LIN {X 0,Y 736.069,Z 312.544,A -85,B 0,C 180,E1 33497.47,E2 33497.47} C_VEL
LIN {X 0,Y 736.097,Z 312.539,A -85,B 0,C 180,E1 33494.554,E2 33494.554} C_VEL
LIN {X 0,Y 736.065,Z 312.54,A -85,B 0,C 180,E1 33491.678,E2 33491.678} C_VEL
LIN {X 0,Y 736.096,Z 312.543,A -85,B 0,C 180,E1 33488.751,E2 33488.751} C_VEL
LIN {X 0,Y 736.064,Z 312.538,A -85,B 0,C 180,E1 33485.848,E2 33485.848} C_VEL
LIN {X 0,Y 736.083,Z 312.544,A -85,B 0,C 180,E1 33483.037,E2 33483.037} C_VEL
LIN {X 0,Y 736.076,Z 312.544,A -85,B 0,C 180,E1 33480.233,E2 33480.233} C_VEL
LIN {X 0,Y 736.068,Z 312.538,A -85,B 0,C 180,E1 33477.353,E2 33477.353} C_VEL
LIN {X 0,Y 736.101,Z 312.54,A -85,B 0,C 180,E1 33474.466,E2 33474.466} C_VEL
LIN {X 0,Y 736.076,Z 312.543,A -85,B 0,C 180,E1 33471.406,E2 33471.406} C_VEL
LIN {X 0,Y 736.093,Z 312.537,A -85,B 0,C 180,E1 33468.561,E2 33468.561} C_VEL
LIN {X 0,Y 736.089,Z 312.533,A -85,B 0,C 180,E1 33465.445,E2 33465.445} C_VEL
LIN {X 0,Y 736.081,Z 312.535,A -85,B 0,C 180,E1 33462.612,E2 33462.612} C_VEL
LIN {X 0,Y 736.096,Z 312.532,A -85,B 0,C 180,E1 33459.568,E2 33459.568} C_VEL
LIN {X 0,Y 736.089,Z 312.722,A -85,B 0,C 180,E1 33458.818,E2 33458.818} C_VEL
LIN {X 0,Y 737.261,Z 315.823,A -85,B 0,C 180,E1 33458.436,E2 33458.436} C_VEL
LIN {X 0,Y 738.594,Z 317.668,A -85,B 0,C 180,E1 33458.143,E2 33458.143} C_VEL
LIN {X 0,Y 740.55,Z 321.622,A -85,B 0,C 180,E1 33457.619,E2 33457.619} C_VEL
LIN {X 0,Y 742.24,Z 325.578,A -85,B 0,C 180,E1 33457.132,E2 33457.132} C_VEL
LIN {X 0,Y 741.769,Z 359.17,A -85,B 0,C 180,E1 33454.617,E2 33454.617} C_VEL
LIN {X 0,Y 741.238,Z 397.411,A -85,B 0,C 180,E1 33451.906,E2 33451.906} C_VEL
LIN {X 0,Y 740.72,Z 434.431,A -85,B 0,C 180,E1 33449.409,E2 33449.409} C_VEL
LIN {X 0,Y 740.274,Z 473.659,A -85,B 0,C 180,E1 33446.867,E2 33446.867} C_VEL
LIN {X 0,Y 740.108,Z 524.032,A -85,B 0,C 180,E1 33443.719,E2 33443.719} C_VEL
LIN {X 0,Y 741.62,Z 532.942,A -85,B 0,C 180,E1 33443.081,E2 33443.081} C_VEL
LIN {X 0,Y 744.357,Z 539.434,A -85,B 0,C 180,E1 33442.518,E2 33442.518} C_VEL
LIN {X 0,Y 746.728,Z 542.692,A -85,B 0,C 180,E1 33442.06,E2 33442.06} C_VEL
LIN {X 0,Y 748.53,Z 544.076,A -85,B 0,C 180,E1 33441.6,E2 33441.6} C_VEL
LIN {X 0,Y 749.609,Z 543.888,A -85,B 0,C 180,E1 33441.165,E2 33441.165} C_VEL
LIN {X 0,Y 749.97,Z 542.102,A -85,B 0,C 180,E1 33440.707,E2 33440.707} C_VEL
LIN {X 0,Y 749.391,Z 538.868,A -85,B 0,C 180,E1 33440.3,E2 33440.3} C_VEL
LIN {X 0,Y 747.937,Z 534.168,A -85,B 0,C 180,E1 33439.966,E2 33439.966} C_VEL
LIN {X 0,Y 745.852,Z 528.342,A -85,B 0,C 180,E1 33439.742,E2 33439.742} C_VEL
LIN {X 0,Y 743.29,Z 519.313,A -85,B 0,C 180,E1 33439.574,E2 33439.574} C_VEL
LIN {X 0,Y 741.804,Z 507.87,A -85,B 0,C 180,E1 33439.476,E2 33439.476} C_VEL
LIN {X 0,Y 741.501,Z 499.262,A -85,B 0,C 180,E1 33439.456,E2 33439.456} C_VEL
LIN {X 0,Y 741.365,Z 321.174,A -85,B 0,C 180,E1 33439.447,E2 33439.447} C_VEL
LIN {X 0,Y 738.994,Z 317.764,A -85,B 0,C 180,E1 33439.289,E2 33439.289} C_VEL
LIN {X 0,Y 736.77,Z 314.896,A -85,B 0,C 180,E1 33439.14,E2 33439.14} C_VEL
LIN {X 0,Y 736.101,Z 312.544,A -85,B 0,C 180,E1 33439.089,E2 33439.089} C_VEL
LIN {X 0,Y 736.094,Z 312.544,A -85,B 0,C 180,E1 33436.15,E2 33436.15} C_VEL
LIN {X 0,Y 736.109,Z 312.612,A -85,B 0,C 180,E1 33435.122,E2 33435.122} C_VEL
LIN {X 0,Y 737.225,Z 315.749,A -85,B 0,C 180,E1 33434.819,E2 33434.819} C_VEL
LIN {X 0,Y 740.443,Z 323.029,A -85,B 0,C 180,E1 33434.076,E2 33434.076} C_VEL
LIN {X 0,Y 740.212,Z 351.073,A -85,B 0,C 180,E1 33432.247,E2 33432.247} C_VEL
LIN {X 0,Y 741.81,Z 357.804,A -85,B 0,C 180,E1 33432.049,E2 33432.049} C_VEL
LIN {X 0,Y 741.13,Z 571.769,A -85,B 0,C 180,E1 33429.415,E2 33429.415} C_VEL
LIN {X 0,Y 740.474,Z 796.533,A -85,B 0,C 180,E1 33426.743,E2 33426.743} C_VEL
LIN {X 0,Y 740.311,Z 833.682,A -85,B 0,C 180,E1 33426.273,E2 33426.273} C_VEL
LIN {X 0,Y 740.077,Z 859.788,A -85,B 0,C 180,E1 33425.793,E2 33425.793} C_VEL
LIN {X 0,Y 739.816,Z 886.294,A -85,B 0,C 180,E1 33425.151,E2 33425.151} C_VEL
LIN {X 0,Y 739.511,Z 913.625,A -85,B 0,C 180,E1 33424.319,E2 33424.319} C_VEL
LIN {X 0,Y 739.096,Z 939.53,A -85,B 0,C 180,E1 33423.361,E2 33423.361} C_VEL
LIN {X 0,Y 738.792,Z 960.718,A -85,B 0,C 180,E1 33422.453,E2 33422.453} C_VEL
LIN {X 0,Y 738.485,Z 982.128,A -85,B 0,C 180,E1 33421.416,E2 33421.416} C_VEL
LIN {X 0,Y 738.067,Z 1007.133,A -85,B 0,C 180,E1 33420.039,E2 33420.039} C_VEL
LIN {X 0,Y 737.724,Z 1028.1,A -85,B 0,C 180,E1 33418.726,E2 33418.726} C_VEL
LIN {X 0,Y 737.437,Z 1048.313,A -85,B 0,C 180,E1 33417.319,E2 33417.319} C_VEL
LIN {X 0,Y 737.073,Z 1069.783,A -85,B 0,C 180,E1 33415.64,E2 33415.64} C_VEL
LIN {X 0,Y 736.848,Z 1086.865,A -85,B 0,C 180,E1 33414.149,E2 33414.149} C_VEL
LIN {X 0,Y 736.632,Z 1104.802,A -85,B 0,C 180,E1 33412.421,E2 33412.421} C_VEL
LIN {X 0,Y 736.415,Z 1121.549,A -85,B 0,C 180,E1 33410.588,E2 33410.588} C_VEL
LIN {X 0,Y 736.271,Z 1134.457,A -85,B 0,C 180,E1 33409.021,E2 33409.021} C_VEL
LIN {X 0,Y 736.172,Z 1147.31,A -85,B 0,C 180,E1 33407.285,E2 33407.285} C_VEL
LIN {X 0,Y 736.041,Z 1161.275,A -85,B 0,C 180,E1 33405.118,E2 33405.118} C_VEL
LIN {X 0,Y 736.01,Z 1170.745,A -85,B 0,C 180,E1 33403.416,E2 33403.416} C_VEL
LIN {X 0,Y 735.948,Z 1178.797,A -85,B 0,C 180,E1 33401.758,E2 33401.758} C_VEL
LIN {X 0,Y 735.942,Z 1186.465,A -85,B 0,C 180,E1 33399.927,E2 33399.927} C_VEL
LIN {X 0,Y 735.927,Z 1193.592,A -85,B 0,C 180,E1 33397.808,E2 33397.808} C_VEL
LIN {X 0,Y 735.918,Z 1199.112,A -85,B 0,C 180,E1 33395.613,E2 33395.613} C_VEL
LIN {X 0,Y 735.915,Z 1202.69,A -85,B 0,C 180,E1 33393.504,E2 33393.504} C_VEL
LIN {X 0,Y 735.913,Z 1204.587,A -85,B 0,C 180,E1 33391.478,E2 33391.478} C_VEL
LIN {X 0,Y 735.89,Z 1204.855,A -85,B 0,C 180,E1 33389.454,E2 33389.454} C_VEL
LIN {X 0,Y 735.906,Z 1203.907,A -85,B 0,C 180,E1 33387.585,E2 33387.585} C_VEL
LIN {X 0,Y 735.907,Z 1201.175,A -85,B 0,C 180,E1 33385.479,E2 33385.479} C_VEL
LIN {X 0,Y 735.916,Z 1196.951,A -85,B 0,C 180,E1 33383.446,E2 33383.446} C_VEL
LIN {X 0,Y 735.932,Z 1191.158,A -85,B 0,C 180,E1 33381.404,E2 33381.404} C_VEL
LIN {X 0,Y 735.931,Z 1183.315,A -85,B 0,C 180,E1 33379.272,E2 33379.272} C_VEL
LIN {X 0,Y 735.999,Z 1173.526,A -85,B 0,C 180,E1 33377.126,E2 33377.126} C_VEL
LIN {X 0,Y 736.041,Z 1164.056,A -85,B 0,C 180,E1 33375.363,E2 33375.363} C_VEL
LIN {X 0,Y 736.096,Z 1154.213,A -85,B 0,C 180,E1 33373.75,E2 33373.75} C_VEL
LIN {X 0,Y 736.202,Z 1143.087,A -85,B 0,C 180,E1 33372.124,E2 33372.124} C_VEL
LIN {X 0,Y 736.376,Z 1127.927,A -85,B 0,C 180,E1 33370.155,E2 33370.155} C_VEL
LIN {X 0,Y 736.521,Z 1112.602,A -85,B 0,C 180,E1 33368.413,E2 33368.413} C_VEL
LIN {X 0,Y 736.686,Z 1097.966,A -85,B 0,C 180,E1 33366.905,E2 33366.905} C_VEL
LIN {X 0,Y 736.984,Z 1079.523,A -85,B 0,C 180,E1 33365.184,E2 33365.184} C_VEL
LIN {X 0,Y 737.237,Z 1059.417,A -85,B 0,C 180,E1 33363.527,E2 33363.527} C_VEL
LIN {X 0,Y 737.575,Z 1039.212,A -85,B 0,C 180,E1 33362.027,E2 33362.027} C_VEL
LIN {X 0,Y 737.942,Z 1015.871,A -85,B 0,C 180,E1 33360.492,E2 33360.492} C_VEL
LIN {X 0,Y 738.235,Z 995.962,A -85,B 0,C 180,E1 33359.324,E2 33359.324} C_VEL
LIN {X 0,Y 738.582,Z 974.073,A -85,B 0,C 180,E1 33358.176,E2 33358.176} C_VEL
LIN {X 0,Y 739.035,Z 947.302,A -85,B 0,C 180,E1 33356.958,E2 33356.958} C_VEL
LIN {X 0,Y 739.329,Z 925.128,A -85,B 0,C 180,E1 33356.09,E2 33356.09} C_VEL
LIN {X 0,Y 739.599,Z 903.358,A -85,B 0,C 180,E1 33355.355,E2 33355.355} C_VEL
LIN {X 0,Y 739.883,Z 879.44,A -85,B 0,C 180,E1 33354.668,E2 33354.668} C_VEL
LIN {X 0,Y 740.16,Z 853.396,A -85,B 0,C 180,E1 33354.075,E2 33354.075} C_VEL
LIN {X 0,Y 740.344,Z 826.293,A -85,B 0,C 180,E1 33353.617,E2 33353.617} C_VEL
LIN {X 0,Y 741.068,Z 590.528,A -85,B 0,C 180,E1 33350.811,E2 33350.811} C_VEL
LIN {X 0,Y 741.708,Z 384.528,A -85,B 0,C 180,E1 33348.284,E2 33348.284} C_VEL
LIN {X 0,Y 741.742,Z 344.371,A -85,B 0,C 180,E1 33347.764,E2 33347.764} C_VEL
LIN {X 0,Y 741.794,Z 322.355,A -85,B 0,C 180,E1 33347.333,E2 33347.333} C_VEL
LIN {X 0,Y 739.204,Z 318.234,A -85,B 0,C 180,E1 33347.065,E2 33347.065} C_VEL
LIN {X 0,Y 736.654,Z 314.64,A -85,B 0,C 180,E1 33346.808,E2 33346.808} C_VEL
LIN {X 0,Y 736.098,Z 312.543,A -85,B 0,C 180,E1 33346.707,E2 33346.707} C_VEL
LIN {X 0,Y 736.075,Z 312.545,A -85,B 0,C 180,E1 33343.836,E2 33343.836} C_VEL
LIN {X 0,Y 736.086,Z 312.538,A -85,B 0,C 180,E1 33340.9,E2 33340.9} C_VEL
LIN {X 0,Y 736.085,Z 312.543,A -85,B 0,C 180,E1 33337.879,E2 33337.879} C_VEL
LIN {X 0,Y 736.095,Z 312.541,A -85,B 0,C 180,E1 33334.976,E2 33334.976} C_VEL
LIN {X 0,Y 736.069,Z 312.534,A -85,B 0,C 180,E1 33332.042,E2 33332.042} C_VEL
LIN {X 0,Y 736.056,Z 312.544,A -85,B 0,C 180,E1 33329.278,E2 33329.278} C_VEL
LIN {X 0,Y 736.088,Z 312.538,A -85,B 0,C 180,E1 33326.372,E2 33326.372} C_VEL
LIN {X 0,Y 736.095,Z 312.542,A -85,B 0,C 180,E1 33323.454,E2 33323.454} C_VEL
LIN {X 0,Y 736.085,Z 312.54,A -85,B 0,C 180,E1 33320.599,E2 33320.599} C_VEL
LIN {X 0,Y 736.079,Z 312.54,A -85,B 0,C 180,E1 33317.523,E2 33317.523} C_VEL
LIN {X 0,Y 736.073,Z 312.544,A -85,B 0,C 180,E1 33314.716,E2 33314.716} C_VEL
LIN {X 0,Y 736.099,Z 312.544,A -85,B 0,C 180,E1 33311.836,E2 33311.836} C_VEL
LIN {X 0,Y 736.088,Z 312.705,A -85,B 0,C 180,E1 33310.973,E2 33310.973} C_VEL
LIN {X 0,Y 736.566,Z 316.487,A -85,B 0,C 180,E1 33310.837,E2 33310.837} C_VEL
LIN {X 0,Y 736.577,Z 395.505,A -85,B 0,C 180,E1 33308.116,E2 33308.116} C_VEL
LIN {X 0,Y 737.021,Z 484.992,A -85,B 0,C 180,E1 33304.903,E2 33304.903} C_VEL
LIN {X 0,Y 737.212,Z 547.222,A -85,B 0,C 180,E1 33302.604,E2 33302.604} C_VEL
LIN {X 0,Y 736.925,Z 624.534,A -85,B 0,C 180,E1 33299.65,E2 33299.65} C_VEL
LIN {X 0,Y 736.633,Z 702.919,A -85,B 0,C 180,E1 33296.69,E2 33296.69} C_VEL
LIN {X 0,Y 736.412,Z 775.104,A -85,B 0,C 180,E1 33294,E2 33294} C_VEL
LIN {X 0,Y 735.417,Z 782.14,A -85,B 0,C 180,E1 33293.756,E2 33293.756} C_VEL
LIN {X 0,Y 729.227,Z 800.996,A -85,B 0,C 180,E1 33293.161,E2 33293.161} C_VEL
LIN {X 0,Y 728.469,Z 807.036,A -85,B 0,C 180,E1 33292.948,E2 33292.948} C_VEL
LIN {X 0,Y 728.406,Z 836.687,A -85,B 0,C 180,E1 33291.863,E2 33291.863} C_VEL
LIN {X 0,Y 728.354,Z 951.855,A -85,B 0,C 180,E1 33290.712,E2 33290.712} C_VEL
LIN {X 0,Y 728.292,Z 966.973,A -85,B 0,C 180,E1 33290.417,E2 33290.417} C_VEL
LIN {X 0,Y 728.231,Z 980.883,A -85,B 0,C 180,E1 33289.998,E2 33289.998} C_VEL
LIN {X 0,Y 728.169,Z 994.335,A -85,B 0,C 180,E1 33289.437,E2 33289.437} C_VEL
LIN {X 0,Y 728.099,Z 1006.123,A -85,B 0,C 180,E1 33288.796,E2 33288.796} C_VEL
LIN {X 0,Y 728.039,Z 1017.779,A -85,B 0,C 180,E1 33287.991,E2 33287.991} C_VEL
LIN {X 0,Y 727.989,Z 1028.194,A -85,B 0,C 180,E1 33287.063,E2 33287.063} C_VEL
LIN {X 0,Y 727.954,Z 1036.705,A -85,B 0,C 180,E1 33286.091,E2 33286.091} C_VEL
LIN {X 0,Y 727.927,Z 1043.764,A -85,B 0,C 180,E1 33285.034,E2 33285.034} C_VEL
LIN {X 0,Y 727.922,Z 1048.588,A -85,B 0,C 180,E1 33284.054,E2 33284.054} C_VEL
LIN {X 0,Y 727.914,Z 1052.009,A -85,B 0,C 180,E1 33283.069,E2 33283.069} C_VEL
LIN {X 0,Y 727.918,Z 1054.107,A -85,B 0,C 180,E1 33282.08,E2 33282.08} C_VEL
LIN {X 0,Y 727.912,Z 1054.957,A -85,B 0,C 180,E1 33280.834,E2 33280.834} C_VEL
LIN {X 0,Y 727.917,Z 1053.969,A -85,B 0,C 180,E1 33279.748,E2 33279.748} C_VEL
LIN {X 0,Y 727.915,Z 1051.955,A -85,B 0,C 180,E1 33278.822,E2 33278.822} C_VEL
LIN {X 0,Y 727.922,Z 1048.382,A -85,B 0,C 180,E1 33277.806,E2 33277.806} C_VEL
LIN {X 0,Y 727.928,Z 1042.753,A -85,B 0,C 180,E1 33276.696,E2 33276.696} C_VEL
LIN {X 0,Y 727.961,Z 1034.947,A -85,B 0,C 180,E1 33275.597,E2 33275.597} C_VEL
LIN {X 0,Y 727.998,Z 1025.932,A -85,B 0,C 180,E1 33274.626,E2 33274.626} C_VEL
LIN {X 0,Y 728.054,Z 1015.423,A -85,B 0,C 180,E1 33273.743,E2 33273.743} C_VEL
LIN {X 0,Y 728.102,Z 1004.453,A -85,B 0,C 180,E1 33273.012,E2 33273.012} C_VEL
LIN {X 0,Y 728.172,Z 991.417,A -85,B 0,C 180,E1 33272.336,E2 33272.336} C_VEL
LIN {X 0,Y 728.241,Z 978.037,A -85,B 0,C 180,E1 33271.815,E2 33271.815} C_VEL
LIN {X 0,Y 728.319,Z 963.352,A -85,B 0,C 180,E1 33271.407,E2 33271.407} C_VEL
LIN {X 0,Y 728.356,Z 949.116,A -85,B 0,C 180,E1 33271.161,E2 33271.161} C_VEL
LIN {X 0,Y 728.37,Z 835.45,A -85,B 0,C 180,E1 33270.02,E2 33270.02} C_VEL
LIN {X 0,Y 728.666,Z 753.979,A -85,B 0,C 180,E1 33266.975,E2 33266.975} C_VEL
LIN {X 0,Y 729.02,Z 675.03,A -85,B 0,C 180,E1 33263.989,E2 33263.989} C_VEL
LIN {X 0,Y 729.395,Z 598.326,A -85,B 0,C 180,E1 33261.053,E2 33261.053} C_VEL
LIN {X 0,Y 729.596,Z 524.571,A -85,B 0,C 180,E1 33258.237,E2 33258.237} C_VEL
LIN {X 0,Y 729.652,Z 467.231,A -85,B 0,C 180,E1 33256.039,E2 33256.039} C_VEL
LIN {X 0,Y 729.688,Z 368.341,A -85,B 0,C 180,E1 33252.337,E2 33252.337} C_VEL
LIN {X 0,Y 730.859,Z 370.392,A -85,B 0,C 180,E1 33252.227,E2 33252.227} C_VEL
LIN {X 0,Y 732.867,Z 370.748,A -85,B 0,C 180,E1 33252.08,E2 33252.08} C_VEL
LIN {X 0,Y 735.681,Z 368.944,A -85,B 0,C 180,E1 33251.905,E2 33251.905} C_VEL
LIN {X 0,Y 734.759,Z 586.79,A -85,B 0,C 180,E1 33249.221,E2 33249.221} C_VEL
LIN {X 0,Y 733.86,Z 799.21,A -85,B 0,C 180,E1 33246.667,E2 33246.667} C_VEL
LIN {X 0,Y 733.597,Z 826.37,A -85,B 0,C 180,E1 33246.19,E2 33246.19} C_VEL
LIN {X 0,Y 733.222,Z 853.624,A -85,B 0,C 180,E1 33245.544,E2 33245.544} C_VEL
LIN {X 0,Y 732.842,Z 877.095,A -85,B 0,C 180,E1 33244.844,E2 33244.844} C_VEL
LIN {X 0,Y 732.463,Z 900.215,A -85,B 0,C 180,E1 33244.035,E2 33244.035} C_VEL
LIN {X 0,Y 731.897,Z 926.739,A -85,B 0,C 180,E1 33242.939,E2 33242.939} C_VEL
LIN {X 0,Y 731.435,Z 948.352,A -85,B 0,C 180,E1 33241.905,E2 33241.905} C_VEL
LIN {X 0,Y 731.017,Z 969.451,A -85,B 0,C 180,E1 33240.768,E2 33240.768} C_VEL
LIN {X 0,Y 730.485,Z 994.26,A -85,B 0,C 180,E1 33239.253,E2 33239.253} C_VEL
LIN {X 0,Y 730.023,Z 1014.652,A -85,B 0,C 180,E1 33237.844,E2 33237.844} C_VEL
LIN {X 0,Y 729.645,Z 1035.627,A -85,B 0,C 180,E1 33236.229,E2 33236.229} C_VEL
LIN {X 0,Y 729.205,Z 1054.965,A -85,B 0,C 180,E1 33234.55,E2 33234.55} C_VEL
LIN {X 0,Y 728.947,Z 1071.789,A -85,B 0,C 180,E1 33232.928,E2 33232.928} C_VEL
LIN {X 0,Y 728.644,Z 1089.728,A -85,B 0,C 180,E1 33230.988,E2 33230.988} C_VEL
LIN {X 0,Y 728.433,Z 1103.44,A -85,B 0,C 180,E1 33229.319,E2 33229.319} C_VEL
LIN {X 0,Y 728.285,Z 1115.085,A -85,B 0,C 180,E1 33227.746,E2 33227.746} C_VEL
LIN {X 0,Y 728.154,Z 1126.005,A -85,B 0,C 180,E1 33226.105,E2 33226.105} C_VEL
LIN {X 0,Y 728.072,Z 1137.953,A -85,B 0,C 180,E1 33224.069,E2 33224.069} C_VEL
LIN {X 0,Y 727.973,Z 1147.868,A -85,B 0,C 180,E1 33222.051,E2 33222.051} C_VEL
LIN {X 0,Y 727.96,Z 1155.96,A -85,B 0,C 180,E1 33220.127,E2 33220.127} C_VEL
LIN {X 0,Y 727.931,Z 1163.268,A -85,B 0,C 180,E1 33217.956,E2 33217.956} C_VEL
LIN {X 0,Y 727.918,Z 1168.668,A -85,B 0,C 180,E1 33215.835,E2 33215.835} C_VEL
LIN {X 0,Y 727.911,Z 1172.316,A -85,B 0,C 180,E1 33213.781,E2 33213.781} C_VEL
LIN {X 0,Y 727.907,Z 1174.457,A -85,B 0,C 180,E1 33211.654,E2 33211.654} C_VEL
LIN {X 0,Y 727.89,Z 1174.896,A -85,B 0,C 180,E1 33209.529,E2 33209.529} C_VEL
LIN {X 0,Y 727.905,Z 1173.955,A -85,B 0,C 180,E1 33207.56,E2 33207.56} C_VEL
LIN {X 0,Y 727.906,Z 1171.129,A -85,B 0,C 180,E1 33205.352,E2 33205.352} C_VEL
LIN {X 0,Y 727.913,Z 1166.846,A -85,B 0,C 180,E1 33203.288,E2 33203.288} C_VEL
LIN {X 0,Y 727.935,Z 1161.042,A -85,B 0,C 180,E1 33201.231,E2 33201.231} C_VEL
LIN {X 0,Y 727.948,Z 1153.183,A -85,B 0,C 180,E1 33199.074,E2 33199.074} C_VEL
LIN {X 0,Y 728.015,Z 1143.346,A -85,B 0,C 180,E1 33196.903,E2 33196.903} C_VEL
LIN {X 0,Y 728.08,Z 1134.313,A -85,B 0,C 180,E1 33195.201,E2 33195.201} C_VEL
LIN {X 0,Y 728.168,Z 1125.023,A -85,B 0,C 180,E1 33193.652,E2 33193.652} C_VEL
LIN {X 0,Y 728.279,Z 1114.459,A -85,B 0,C 180,E1 33192.075,E2 33192.075} C_VEL
LIN {X 0,Y 728.441,Z 1102.862,A -85,B 0,C 180,E1 33190.517,E2 33190.517} C_VEL
LIN {X 0,Y 728.672,Z 1087.897,A -85,B 0,C 180,E1 33188.707,E2 33188.707} C_VEL
LIN {X 0,Y 728.949,Z 1070.149,A -85,B 0,C 180,E1 33186.818,E2 33186.818} C_VEL
LIN {X 0,Y 729.229,Z 1054.094,A -85,B 0,C 180,E1 33185.28,E2 33185.28} C_VEL
LIN {X 0,Y 729.666,Z 1034.091,A -85,B 0,C 180,E1 33183.555,E2 33183.555} C_VEL
LIN {X 0,Y 730.047,Z 1013.488,A -85,B 0,C 180,E1 33181.981,E2 33181.981} C_VEL
LIN {X 0,Y 730.574,Z 991.628,A -85,B 0,C 180,E1 33180.483,E2 33180.483} C_VEL
LIN {X 0,Y 731.023,Z 968.665,A -85,B 0,C 180,E1 33179.097,E2 33179.097} C_VEL
LIN {X 0,Y 731.444,Z 947.651,A -85,B 0,C 180,E1 33177.969,E2 33177.969} C_VEL
LIN {X 0,Y 732.037,Z 922.741,A -85,B 0,C 180,E1 33176.791,E2 33176.791} C_VEL
LIN {X 0,Y 732.493,Z 897.647,A -85,B 0,C 180,E1 33175.78,E2 33175.78} C_VEL
LIN {X 0,Y 732.852,Z 876.27,A -85,B 0,C 180,E1 33175.039,E2 33175.039} C_VEL
LIN {X 0,Y 733.234,Z 852.804,A -85,B 0,C 180,E1 33174.344,E2 33174.344} C_VEL
LIN {X 0,Y 733.622,Z 825.243,A -85,B 0,C 180,E1 33173.697,E2 33173.697} C_VEL
LIN {X 0,Y 733.872,Z 797.791,A -85,B 0,C 180,E1 33173.222,E2 33173.222} C_VEL
LIN {X 0,Y 734.863,Z 561.125,A -85,B 0,C 180,E1 33170.378,E2 33170.378} C_VEL
LIN {X 0,Y 735.738,Z 350.961,A -85,B 0,C 180,E1 33167.777,E2 33167.777} C_VEL
LIN {X 0,Y 735.645,Z 329.251,A -85,B 0,C 180,E1 33167.49,E2 33167.49} C_VEL
LIN {X 0,Y 734.468,Z 325.955,A -85,B 0,C 180,E1 33167.363,E2 33167.363} C_VEL
LIN {X 0,Y 731.048,Z 320.731,A -85,B 0,C 180,E1 33167.033,E2 33167.033} C_VEL
LIN {X 0,Y 728.172,Z 313.695,A -85,B 0,C 180,E1 33166.311,E2 33166.311} C_VEL
LIN {X 0,Y 728.141,Z 313.533,A -85,B 0,C 180,E1 33163.415,E2 33163.415} C_VEL
LIN {X 0,Y 728.149,Z 313.534,A -85,B 0,C 180,E1 33160.472,E2 33160.472} C_VEL
LIN {X 0,Y 728.159,Z 313.53,A -85,B 0,C 180,E1 33157.468,E2 33157.468} C_VEL
LIN {X 0,Y 728.155,Z 313.527,A -85,B 0,C 180,E1 33154.455,E2 33154.455} C_VEL
LIN {X 0,Y 728.162,Z 313.53,A -85,B 0,C 180,E1 33151.361,E2 33151.361} C_VEL
LIN {X 0,Y 728.144,Z 313.527,A -85,B 0,C 180,E1 33148.457,E2 33148.457} C_VEL
LIN {X 0,Y 728.136,Z 313.529,A -85,B 0,C 180,E1 33145.543,E2 33145.543} C_VEL
LIN {X 0,Y 728.153,Z 313.534,A -85,B 0,C 180,E1 33142.669,E2 33142.669} C_VEL
LIN {X 0,Y 728.126,Z 313.525,A -85,B 0,C 180,E1 33139.828,E2 33139.828} C_VEL
LIN {X 0,Y 728.16,Z 313.529,A -85,B 0,C 180,E1 33136.925,E2 33136.925} C_VEL
LIN {X 0,Y 728.126,Z 313.532,A -85,B 0,C 180,E1 33133.986,E2 33133.986} C_VEL
LIN {X 0,Y 728.156,Z 313.522,A -85,B 0,C 180,E1 33131.084,E2 33131.084} C_VEL
LIN {X 0,Y 728.126,Z 313.533,A -85,B 0,C 180,E1 33128.131,E2 33128.131} C_VEL
LIN {X 0,Y 728.152,Z 313.525,A -85,B 0,C 180,E1 33125.279,E2 33125.279} C_VEL
LIN {X 0,Y 728.148,Z 313.525,A -85,B 0,C 180,E1 33122.361,E2 33122.361} C_VEL
LIN {X 0,Y 728.159,Z 313.533,A -85,B 0,C 180,E1 33119.371,E2 33119.371} C_VEL
LIN {X 0,Y 728.159,Z 313.525,A -85,B 0,C 180,E1 33116.3,E2 33116.3} C_VEL
LIN {X 0,Y 728.152,Z 313.521,A -85,B 0,C 180,E1 33113.376,E2 33113.376} C_VEL
LIN {X 0,Y 728.158,Z 313.529,A -85,B 0,C 180,E1 33110.276,E2 33110.276} C_VEL
LIN {X 0,Y 728.14,Z 313.533,A -85,B 0,C 180,E1 33107.388,E2 33107.388} C_VEL
LIN {X 0,Y 728.128,Z 313.528,A -85,B 0,C 180,E1 33104.549,E2 33104.549} C_VEL
LIN {X 0,Y 728.152,Z 313.516,A -85,B 0,C 180,E1 33101.672,E2 33101.672} C_VEL
LIN {X 0,Y 728.174,Z 313.651,A -85,B 0,C 180,E1 33099.629,E2 33099.629} C_VEL
LIN {X 0,Y 729.533,Z 317.128,A -85,B 0,C 180,E1 33099.181,E2 33099.181} C_VEL
LIN {X 0,Y 730.704,Z 318.85,A -85,B 0,C 180,E1 33098.907,E2 33098.907} C_VEL
LIN {X 0,Y 732.665,Z 322.642,A -85,B 0,C 180,E1 33098.378,E2 33098.378} C_VEL
LIN {X 0,Y 736.388,Z 330.094,A -85,B 0,C 180,E1 33097.381,E2 33097.381} C_VEL
LIN {X 0,Y 735.748,Z 363.429,A -85,B 0,C 180,E1 33094.869,E2 33094.869} C_VEL
LIN {X 0,Y 735.023,Z 402.256,A -85,B 0,C 180,E1 33092.098,E2 33092.098} C_VEL
LIN {X 0,Y 734.331,Z 439.535,A -85,B 0,C 180,E1 33089.567,E2 33089.567} C_VEL
LIN {X 0,Y 733.725,Z 478.669,A -85,B 0,C 180,E1 33087.015,E2 33087.015} C_VEL
LIN {X 0,Y 733.362,Z 526.382,A -85,B 0,C 180,E1 33084.01,E2 33084.01} C_VEL
LIN {X 0,Y 734.814,Z 536.073,A -85,B 0,C 180,E1 33083.318,E2 33083.318} C_VEL
LIN {X 0,Y 737.58,Z 543.354,A -85,B 0,C 180,E1 33082.701,E2 33082.701} C_VEL
LIN {X 0,Y 740.832,Z 548.005,A -85,B 0,C 180,E1 33082.211,E2 33082.211} C_VEL
LIN {X 0,Y 743.498,Z 550.407,A -85,B 0,C 180,E1 33081.754,E2 33081.754} C_VEL
LIN {X 0,Y 745.358,Z 551.113,A -85,B 0,C 180,E1 33081.308,E2 33081.308} C_VEL
LIN {X 0,Y 746.449,Z 550.425,A -85,B 0,C 180,E1 33080.856,E2 33080.856} C_VEL
LIN {X 0,Y 746.623,Z 548.245,A -85,B 0,C 180,E1 33080.397,E2 33080.397} C_VEL
LIN {X 0,Y 745.744,Z 544.729,A -85,B 0,C 180,E1 33079.99,E2 33079.99} C_VEL
LIN {X 0,Y 743.897,Z 539.969,A -85,B 0,C 180,E1 33079.664,E2 33079.664} C_VEL
LIN {X 0,Y 741.128,Z 533.733,A -85,B 0,C 180,E1 33079.431,E2 33079.431} C_VEL
LIN {X 0,Y 738.095,Z 524.389,A -85,B 0,C 180,E1 33079.229,E2 33079.229} C_VEL
LIN {X 0,Y 736.155,Z 513.061,A -85,B 0,C 180,E1 33079.099,E2 33079.099} C_VEL
LIN {X 0,Y 735.441,Z 499.366,A -85,B 0,C 180,E1 33079.051,E2 33079.051} C_VEL
LIN {X 0,Y 735.25,Z 324.085,A -85,B 0,C 180,E1 33079.038,E2 33079.038} C_VEL
LIN {X 0,Y 732.196,Z 320.203,A -85,B 0,C 180,E1 33078.83,E2 33078.83} C_VEL
LIN {X 0,Y 731.068,Z 318.786,A -85,B 0,C 180,E1 33078.753,E2 33078.753} C_VEL
LIN {X 0,Y 728.815,Z 315.939,A -85,B 0,C 180,E1 33078.597,E2 33078.597} C_VEL
LIN {X 0,Y 728.118,Z 313.536,A -85,B 0,C 180,E1 33078.537,E2 33078.537} C_VEL
LIN {X 0,Y 728.145,Z 313.562,A -85,B 0,C 180,E1 33075.688,E2 33075.688} C_VEL
LIN {X 0,Y 729.546,Z 317.136,A -85,B 0,C 180,E1 33075.323,E2 33075.323} C_VEL
LIN {X 0,Y 733.95,Z 326.84,A -85,B 0,C 180,E1 33074.307,E2 33074.307} C_VEL
LIN {X 0,Y 733.707,Z 351.153,A -85,B 0,C 180,E1 33072.709,E2 33072.709} C_VEL
LIN {X 0,Y 735.844,Z 360.026,A -85,B 0,C 180,E1 33072.441,E2 33072.441} C_VEL
LIN {X 0,Y 734.932,Z 573.195,A -85,B 0,C 180,E1 33069.796,E2 33069.796} C_VEL
LIN {X 0,Y 734.049,Z 797.747,A -85,B 0,C 180,E1 33067.104,E2 33067.104} C_VEL
LIN {X 0,Y 733.835,Z 834.187,A -85,B 0,C 180,E1 33066.637,E2 33066.637} C_VEL
LIN {X 0,Y 733.52,Z 860.604,A -85,B 0,C 180,E1 33066.145,E2 33066.145} C_VEL
LIN {X 0,Y 733.164,Z 887.168,A -85,B 0,C 180,E1 33065.492,E2 33065.492} C_VEL
LIN {X 0,Y 732.728,Z 915.143,A -85,B 0,C 180,E1 33064.627,E2 33064.627} C_VEL
LIN {X 0,Y 732.2,Z 940.657,A -85,B 0,C 180,E1 33063.67,E2 33063.67} C_VEL
LIN {X 0,Y 731.79,Z 961.717,A -85,B 0,C 180,E1 33062.755,E2 33062.755} C_VEL
LIN {X 0,Y 731.346,Z 985.68,A -85,B 0,C 180,E1 33061.575,E2 33061.575} C_VEL
LIN {X 0,Y 730.753,Z 1010.088,A -85,B 0,C 180,E1 33060.187,E2 33060.187} C_VEL
LIN {X 0,Y 730.346,Z 1029.589,A -85,B 0,C 180,E1 33058.943,E2 33058.943} C_VEL
LIN {X 0,Y 729.936,Z 1051.281,A -85,B 0,C 180,E1 33057.403,E2 33057.403} C_VEL
LIN {X 0,Y 729.458,Z 1071.818,A -85,B 0,C 180,E1 33055.753,E2 33055.753} C_VEL
LIN {X 0,Y 729.165,Z 1089.197,A -85,B 0,C 180,E1 33054.204,E2 33054.204} C_VEL
LIN {X 0,Y 728.818,Z 1107.942,A -85,B 0,C 180,E1 33052.334,E2 33052.334} C_VEL
LIN {X 0,Y 728.594,Z 1122.261,A -85,B 0,C 180,E1 33050.735,E2 33050.735} C_VEL
LIN {X 0,Y 728.401,Z 1135.105,A -85,B 0,C 180,E1 33049.151,E2 33049.151} C_VEL
LIN {X 0,Y 728.259,Z 1148.924,A -85,B 0,C 180,E1 33047.25,E2 33047.25} C_VEL
LIN {X 0,Y 728.097,Z 1161.742,A -85,B 0,C 180,E1 33045.205,E2 33045.205} C_VEL
LIN {X 0,Y 728.041,Z 1171.082,A -85,B 0,C 180,E1 33043.5,E2 33043.5} C_VEL
LIN {X 0,Y 727.967,Z 1179.157,A -85,B 0,C 180,E1 33041.808,E2 33041.808} C_VEL
LIN {X 0,Y 727.953,Z 1186.729,A -85,B 0,C 180,E1 33039.965,E2 33039.965} C_VEL
LIN {X 0,Y 727.93,Z 1193.59,A -85,B 0,C 180,E1 33037.894,E2 33037.894} C_VEL
LIN {X 0,Y 727.919,Z 1199.113,A -85,B 0,C 180,E1 33035.675,E2 33035.675} C_VEL
LIN {X 0,Y 727.915,Z 1202.691,A -85,B 0,C 180,E1 33033.543,E2 33033.543} C_VEL
LIN {X 0,Y 727.912,Z 1204.588,A -85,B 0,C 180,E1 33031.495,E2 33031.495} C_VEL
LIN {X 0,Y 727.89,Z 1204.857,A -85,B 0,C 180,E1 33029.448,E2 33029.448} C_VEL
LIN {X 0,Y 727.906,Z 1203.907,A -85,B 0,C 180,E1 33027.558,E2 33027.558} C_VEL
LIN {X 0,Y 727.907,Z 1201.174,A -85,B 0,C 180,E1 33025.429,E2 33025.429} C_VEL
LIN {X 0,Y 727.917,Z 1196.951,A -85,B 0,C 180,E1 33023.373,E2 33023.373} C_VEL
LIN {X 0,Y 727.936,Z 1191.158,A -85,B 0,C 180,E1 33021.309,E2 33021.309} C_VEL
LIN {X 0,Y 727.947,Z 1183.291,A -85,B 0,C 180,E1 33019.147,E2 33019.147} C_VEL
LIN {X 0,Y 728.028,Z 1173.53,A -85,B 0,C 180,E1 33016.982,E2 33016.982} C_VEL
LIN {X 0,Y 728.082,Z 1164.058,A -85,B 0,C 180,E1 33015.2,E2 33015.2} C_VEL
LIN {X 0,Y 728.179,Z 1154.216,A -85,B 0,C 180,E1 33013.568,E2 33013.568} C_VEL
LIN {X 0,Y 728.331,Z 1142.278,A -85,B 0,C 180,E1 33011.809,E2 33011.809} C_VEL
LIN {X 0,Y 728.549,Z 1125.797,A -85,B 0,C 180,E1 33009.682,E2 33009.682} C_VEL
LIN {X 0,Y 728.762,Z 1111.477,A -85,B 0,C 180,E1 33008.049,E2 33008.049} C_VEL
LIN {X 0,Y 728.989,Z 1097.114,A -85,B 0,C 180,E1 33006.561,E2 33006.561} C_VEL
LIN {X 0,Y 729.396,Z 1077.874,A -85,B 0,C 180,E1 33004.764,E2 33004.764} C_VEL
LIN {X 0,Y 729.717,Z 1059.064,A -85,B 0,C 180,E1 33003.204,E2 33003.204} C_VEL
LIN {X 0,Y 730.219,Z 1038.008,A -85,B 0,C 180,E1 33001.63,E2 33001.63} C_VEL
LIN {X 0,Y 730.667,Z 1015.146,A -85,B 0,C 180,E1 33000.124,E2 33000.124} C_VEL
LIN {X 0,Y 731.08,Z 994.627,A -85,B 0,C 180,E1 32998.915,E2 32998.915} C_VEL
LIN {X 0,Y 731.638,Z 971.388,A -85,B 0,C 180,E1 32997.699,E2 32997.699} C_VEL
LIN {X 0,Y 732.137,Z 946.193,A -85,B 0,C 180,E1 32996.559,E2 32996.559} C_VEL
LIN {X 0,Y 732.532,Z 923.503,A -85,B 0,C 180,E1 32995.671,E2 32995.671} C_VEL
LIN {X 0,Y 732.922,Z 900.437,A -85,B 0,C 180,E1 32994.898,E2 32994.898} C_VEL
LIN {X 0,Y 733.353,Z 874.699,A -85,B 0,C 180,E1 32994.181,E2 32994.181} C_VEL
LIN {X 0,Y 733.694,Z 847.458,A -85,B 0,C 180,E1 32993.59,E2 32993.59} C_VEL
LIN {X 0,Y 733.937,Z 820.871,A -85,B 0,C 180,E1 32993.173,E2 32993.173} C_VEL
LIN {X 0,Y 734.851,Z 591.928,A -85,B 0,C 180,E1 32990.432,E2 32990.432} C_VEL
LIN {X 0,Y 735.716,Z 386.016,A -85,B 0,C 180,E1 32987.886,E2 32987.886} C_VEL
LIN {X 0,Y 735.755,Z 345.262,A -85,B 0,C 180,E1 32987.357,E2 32987.357} C_VEL
LIN {X 0,Y 735.693,Z 326.332,A -85,B 0,C 180,E1 32986.973,E2 32986.973} C_VEL
LIN {X 0,Y 733.104,Z 322.381,A -85,B 0,C 180,E1 32986.704,E2 32986.704} C_VEL
LIN {X 0,Y 730.787,Z 318.546,A -85,B 0,C 180,E1 32986.455,E2 32986.455} C_VEL
LIN {X 0,Y 728.669,Z 315.599,A -85,B 0,C 180,E1 32986.235,E2 32986.235} C_VEL
LIN {X 0,Y 728.121,Z 313.536,A -85,B 0,C 180,E1 32986.134,E2 32986.134} C_VEL
LIN {X 0,Y 728.117,Z 313.535,A -85,B 0,C 180,E1 32983.41,E2 32983.41} C_VEL
LIN {X 0,Y 728.161,Z 313.521,A -85,B 0,C 180,E1 32980.47,E2 32980.47} C_VEL
LIN {X 0,Y 728.154,Z 313.522,A -85,B 0,C 180,E1 32977.568,E2 32977.568} C_VEL
LIN {X 0,Y 728.158,Z 313.529,A -85,B 0,C 180,E1 32974.522,E2 32974.522} C_VEL
LIN {X 0,Y 728.137,Z 313.518,A -85,B 0,C 180,E1 32971.455,E2 32971.455} C_VEL
LIN {X 0,Y 728.164,Z 313.533,A -85,B 0,C 180,E1 32968.546,E2 32968.546} C_VEL
LIN {X 0,Y 728.121,Z 313.515,A -85,B 0,C 180,E1 32965.631,E2 32965.631} C_VEL
LIN {X 0,Y 728.12,Z 313.533,A -85,B 0,C 180,E1 32962.955,E2 32962.955} C_VEL
LIN {X 0,Y 728.161,Z 313.527,A -85,B 0,C 180,E1 32959.91,E2 32959.91} C_VEL
LIN {X 0,Y 728.151,Z 313.53,A -85,B 0,C 180,E1 32956.925,E2 32956.925} C_VEL
LIN {X 0,Y 728.16,Z 313.528,A -85,B 0,C 180,E1 32953.872,E2 32953.872} C_VEL
LIN {X 0,Y 728.157,Z 313.772,A -85,B 0,C 180,E1 32951.094,E2 32951.094} C_VEL
LIN {X 0,Y 728.775,Z 317.593,A -85,B 0,C 180,E1 32950.954,E2 32950.954} C_VEL
LIN {X 0,Y 728.813,Z 394.302,A -85,B 0,C 180,E1 32948.322,E2 32948.322} C_VEL
LIN {X 0,Y 729.177,Z 477.201,A -85,B 0,C 180,E1 32945.35,E2 32945.35} C_VEL
LIN {X 0,Y 729.424,Z 541.368,A -85,B 0,C 180,E1 32942.986,E2 32942.986} C_VEL
LIN {X 0,Y 729.352,Z 610.534,A -85,B 0,C 180,E1 32940.393,E2 32940.393} C_VEL
LIN {X 0,Y 728.947,Z 689.631,A -85,B 0,C 180,E1 32937.366,E2 32937.366} C_VEL
LIN {X 0,Y 728.605,Z 768.012,A -85,B 0,C 180,E1 32934.408,E2 32934.408} C_VEL
LIN {X 0,Y 728.469,Z 807.036,A -85,B 0,C 180,E1 32932.948,E2 32932.948} C_VEL
LIN {X 0,Y 727.538,Z 814.881,A -85,B 0,C 180,E1 32932.677,E2 32932.677} C_VEL
LIN {X 0,Y 723.853,Z 826.587,A -85,B 0,C 180,E1 32932.291,E2 32932.291} C_VEL
LIN {X 0,Y 720.989,Z 835.59,A -85,B 0,C 180,E1 32932.02,E2 32932.02} C_VEL
LIN {X 0,Y 720.594,Z 839.219,A -85,B 0,C 180,E1 32931.958,E2 32931.958} C_VEL
LIN {X 0,Y 720.47,Z 952.195,A -85,B 0,C 180,E1 32930.816,E2 32930.816} C_VEL
LIN {X 0,Y 720.39,Z 967.287,A -85,B 0,C 180,E1 32930.513,E2 32930.513} C_VEL
LIN {X 0,Y 720.316,Z 979.963,A -85,B 0,C 180,E1 32930.129,E2 32930.129} C_VEL
LIN {X 0,Y 720.246,Z 992.854,A -85,B 0,C 180,E1 32929.603,E2 32929.603} C_VEL
LIN {X 0,Y 720.149,Z 1005.641,A -85,B 0,C 180,E1 32928.913,E2 32928.913} C_VEL
LIN {X 0,Y 720.076,Z 1017.381,A -85,B 0,C 180,E1 32928.1,E2 32928.1} C_VEL
LIN {X 0,Y 720.008,Z 1028.19,A -85,B 0,C 180,E1 32927.131,E2 32927.131} C_VEL
LIN {X 0,Y 719.966,Z 1036.448,A -85,B 0,C 180,E1 32926.18,E2 32926.18} C_VEL
LIN {X 0,Y 719.93,Z 1043.603,A -85,B 0,C 180,E1 32925.111,E2 32925.111} C_VEL
LIN {X 0,Y 719.923,Z 1048.803,A -85,B 0,C 180,E1 32924.038,E2 32924.038} C_VEL
LIN {X 0,Y 719.915,Z 1052.147,A -85,B 0,C 180,E1 32923.042,E2 32923.042} C_VEL
LIN {X 0,Y 719.915,Z 1054.46,A -85,B 0,C 180,E1 32921.874,E2 32921.874} C_VEL
LIN {X 0,Y 719.909,Z 1054.883,A -85,B 0,C 180,E1 32920.697,E2 32920.697} C_VEL
LIN {X 0,Y 719.919,Z 1053.883,A -85,B 0,C 180,E1 32919.682,E2 32919.682} C_VEL
LIN {X 0,Y 719.913,Z 1051.798,A -85,B 0,C 180,E1 32918.742,E2 32918.742} C_VEL
LIN {X 0,Y 719.925,Z 1047.968,A -85,B 0,C 180,E1 32917.668,E2 32917.668} C_VEL
LIN {X 0,Y 719.938,Z 1041.848,A -85,B 0,C 180,E1 32916.509,E2 32916.509} C_VEL
LIN {X 0,Y 719.971,Z 1035.051,A -85,B 0,C 180,E1 32915.552,E2 32915.552} C_VEL
LIN {X 0,Y 720.019,Z 1026.284,A -85,B 0,C 180,E1 32914.589,E2 32914.589} C_VEL
LIN {X 0,Y 720.086,Z 1016.01,A -85,B 0,C 180,E1 32913.707,E2 32913.707} C_VEL
LIN {X 0,Y 720.153,Z 1004.589,A -85,B 0,C 180,E1 32912.931,E2 32912.931} C_VEL
LIN {X 0,Y 720.245,Z 991.138,A -85,B 0,C 180,E1 32912.228,E2 32912.228} C_VEL
LIN {X 0,Y 720.332,Z 977.879,A -85,B 0,C 180,E1 32911.709,E2 32911.709} C_VEL
LIN {X 0,Y 720.427,Z 963.183,A -85,B 0,C 180,E1 32911.297,E2 32911.297} C_VEL
LIN {X 0,Y 720.471,Z 948.776,A -85,B 0,C 180,E1 32911.048,E2 32911.048} C_VEL
LIN {X 0,Y 720.493,Z 835.77,A -85,B 0,C 180,E1 32909.911,E2 32909.911} C_VEL
LIN {X 0,Y 720.863,Z 754.433,A -85,B 0,C 180,E1 32906.838,E2 32906.838} C_VEL
LIN {X 0,Y 721.307,Z 675.959,A -85,B 0,C 180,E1 32903.837,E2 32903.837} C_VEL
LIN {X 0,Y 721.661,Z 598.689,A -85,B 0,C 180,E1 32900.887,E2 32900.887} C_VEL
LIN {X 0,Y 721.962,Z 525.159,A -85,B 0,C 180,E1 32898.05,E2 32898.05} C_VEL
LIN {X 0,Y 722.013,Z 481.208,A -85,B 0,C 180,E1 32896.367,E2 32896.367} C_VEL
LIN {X 0,Y 722.036,Z 383.601,A -85,B 0,C 180,E1 32892.691,E2 32892.691} C_VEL
LIN {X 0,Y 723.307,Z 385.853,A -85,B 0,C 180,E1 32892.568,E2 32892.568} C_VEL
LIN {X 0,Y 724.935,Z 386.204,A -85,B 0,C 180,E1 32892.445,E2 32892.445} C_VEL
LIN {X 0,Y 727.462,Z 384.664,A -85,B 0,C 180,E1 32892.284,E2 32892.284} C_VEL
LIN {X 0,Y 729.65,Z 382.251,A -85,B 0,C 180,E1 32892.159,E2 32892.159} C_VEL
LIN {X 0,Y 728.488,Z 599.303,A -85,B 0,C 180,E1 32889.468,E2 32889.468} C_VEL
LIN {X 0,Y 727.427,Z 799.248,A -85,B 0,C 180,E1 32887.046,E2 32887.046} C_VEL
LIN {X 0,Y 727.099,Z 826.317,A -85,B 0,C 180,E1 32886.567,E2 32886.567} C_VEL
LIN {X 0,Y 726.625,Z 853.523,A -85,B 0,C 180,E1 32885.919,E2 32885.919} C_VEL
LIN {X 0,Y 726.15,Z 877.119,A -85,B 0,C 180,E1 32885.213,E2 32885.213} C_VEL
LIN {X 0,Y 725.646,Z 901.467,A -85,B 0,C 180,E1 32884.352,E2 32884.352} C_VEL
LIN {X 0,Y 724.948,Z 927.752,A -85,B 0,C 180,E1 32883.248,E2 32883.248} C_VEL
LIN {X 0,Y 724.364,Z 949.45,A -85,B 0,C 180,E1 32882.197,E2 32882.197} C_VEL
LIN {X 0,Y 723.809,Z 971.845,A -85,B 0,C 180,E1 32880.97,E2 32880.97} C_VEL
LIN {X 0,Y 723.148,Z 995.599,A -85,B 0,C 180,E1 32879.488,E2 32879.488} C_VEL
LIN {X 0,Y 722.565,Z 1016.656,A -85,B 0,C 180,E1 32878.009,E2 32878.009} C_VEL
LIN {X 0,Y 722.026,Z 1038.745,A -85,B 0,C 180,E1 32876.261,E2 32876.261} C_VEL
LIN {X 0,Y 721.523,Z 1057.204,A -85,B 0,C 180,E1 32874.62,E2 32874.62} C_VEL
LIN {X 0,Y 721.14,Z 1075.946,A -85,B 0,C 180,E1 32872.759,E2 32872.759} C_VEL
LIN {X 0,Y 720.806,Z 1091.865,A -85,B 0,C 180,E1 32870.972,E2 32870.972} C_VEL
LIN {X 0,Y 720.563,Z 1104.734,A -85,B 0,C 180,E1 32869.37,E2 32869.37} C_VEL
LIN {X 0,Y 720.37,Z 1117.417,A -85,B 0,C 180,E1 32867.614,E2 32867.614} C_VEL
LIN {X 0,Y 720.177,Z 1131.469,A -85,B 0,C 180,E1 32865.379,E2 32865.379} C_VEL
LIN {X 0,Y 720.068,Z 1140.83,A -85,B 0,C 180,E1 32863.655,E2 32863.655} C_VEL
LIN {X 0,Y 719.99,Z 1148.586,A -85,B 0,C 180,E1 32862.024,E2 32862.024} C_VEL
LIN {X 0,Y 719.971,Z 1156.256,A -85,B 0,C 180,E1 32860.16,E2 32860.16} C_VEL
LIN {X 0,Y 719.935,Z 1163.451,A -85,B 0,C 180,E1 32857.984,E2 32857.984} C_VEL
LIN {X 0,Y 719.921,Z 1169.013,A -85,B 0,C 180,E1 32855.74,E2 32855.74} C_VEL
LIN {X 0,Y 719.912,Z 1172.518,A -85,B 0,C 180,E1 32853.664,E2 32853.664} C_VEL
LIN {X 0,Y 719.909,Z 1174.553,A -85,B 0,C 180,E1 32851.513,E2 32851.513} C_VEL
LIN {X 0,Y 719.891,Z 1174.877,A -85,B 0,C 180,E1 32849.444,E2 32849.444} C_VEL
LIN {X 0,Y 719.906,Z 1173.876,A -85,B 0,C 180,E1 32847.454,E2 32847.454} C_VEL
LIN {X 0,Y 719.909,Z 1171,A -85,B 0,C 180,E1 32845.221,E2 32845.221} C_VEL
LIN {X 0,Y 719.915,Z 1166.666,A -85,B 0,C 180,E1 32843.141,E2 32843.141} C_VEL
LIN {X 0,Y 719.94,Z 1161.037,A -85,B 0,C 180,E1 32841.133,E2 32841.133} C_VEL
LIN {X 0,Y 719.97,Z 1153.182,A -85,B 0,C 180,E1 32838.952,E2 32838.952} C_VEL
LIN {X 0,Y 720.052,Z 1143.344,A -85,B 0,C 180,E1 32836.756,E2 32836.756} C_VEL
LIN {X 0,Y 720.126,Z 1134.316,A -85,B 0,C 180,E1 32835.034,E2 32835.034} C_VEL
LIN {X 0,Y 720.251,Z 1125.019,A -85,B 0,C 180,E1 32833.467,E2 32833.467} C_VEL
LIN {X 0,Y 720.393,Z 1114.565,A -85,B 0,C 180,E1 32831.887,E2 32831.887} C_VEL
LIN {X 0,Y 720.585,Z 1103.503,A -85,B 0,C 180,E1 32830.38,E2 32830.38} C_VEL
LIN {X 0,Y 720.84,Z 1089.791,A -85,B 0,C 180,E1 32828.691,E2 32828.691} C_VEL
LIN {X 0,Y 721.214,Z 1071.854,A -85,B 0,C 180,E1 32826.728,E2 32826.728} C_VEL
LIN {X 0,Y 721.587,Z 1055.024,A -85,B 0,C 180,E1 32825.088,E2 32825.088} C_VEL
LIN {X 0,Y 722.098,Z 1035.825,A -85,B 0,C 180,E1 32823.402,E2 32823.402} C_VEL
LIN {X 0,Y 722.616,Z 1014.696,A -85,B 0,C 180,E1 32821.758,E2 32821.758} C_VEL
LIN {X 0,Y 723.275,Z 992.303,A -85,B 0,C 180,E1 32820.201,E2 32820.201} C_VEL
LIN {X 0,Y 723.851,Z 968.824,A -85,B 0,C 180,E1 32818.766,E2 32818.766} C_VEL
LIN {X 0,Y 724.414,Z 947.646,A -85,B 0,C 180,E1 32817.621,E2 32817.621} C_VEL
LIN {X 0,Y 725.139,Z 922.732,A -85,B 0,C 180,E1 32816.433,E2 32816.433} C_VEL
LIN {X 0,Y 725.705,Z 897.637,A -85,B 0,C 180,E1 32815.414,E2 32815.414} C_VEL
LIN {X 0,Y 726.167,Z 875.523,A -85,B 0,C 180,E1 32814.645,E2 32814.645} C_VEL
LIN {X 0,Y 726.654,Z 851.677,A -85,B 0,C 180,E1 32813.94,E2 32813.94} C_VEL
LIN {X 0,Y 727.131,Z 824.08,A -85,B 0,C 180,E1 32813.298,E2 32813.298} C_VEL
LIN {X 0,Y 727.445,Z 797.372,A -85,B 0,C 180,E1 32812.838,E2 32812.838} C_VEL
LIN {X 0,Y 728.675,Z 563.664,A -85,B 0,C 180,E1 32810.007,E2 32810.007} C_VEL
LIN {X 0,Y 729.787,Z 352.832,A -85,B 0,C 180,E1 32807.377,E2 32807.377} C_VEL
LIN {X 0,Y 729.737,Z 331.49,A -85,B 0,C 180,E1 32807.093,E2 32807.093} C_VEL
LIN {X 0,Y 722.632,Z 320.813,A -85,B 0,C 180,E1 32806.416,E2 32806.416} C_VEL
LIN {X 0,Y 720.223,Z 314.52,A -85,B 0,C 180,E1 32805.756,E2 32805.756} C_VEL
LIN {X 0,Y 720.213,Z 314.522,A -85,B 0,C 180,E1 32802.744,E2 32802.744} C_VEL
LIN {X 0,Y 720.218,Z 314.519,A -85,B 0,C 180,E1 32799.727,E2 32799.727} C_VEL
LIN {X 0,Y 720.215,Z 314.519,A -85,B 0,C 180,E1 32796.753,E2 32796.753} C_VEL
LIN {X 0,Y 720.197,Z 314.511,A -85,B 0,C 180,E1 32793.83,E2 32793.83} C_VEL
LIN {X 0,Y 720.218,Z 314.52,A -85,B 0,C 180,E1 32790.909,E2 32790.909} C_VEL
LIN {X 0,Y 720.186,Z 314.52,A -85,B 0,C 180,E1 32788.077,E2 32788.077} C_VEL
LIN {X 0,Y 720.218,Z 314.509,A -85,B 0,C 180,E1 32785.14,E2 32785.14} C_VEL
LIN {X 0,Y 720.188,Z 314.523,A -85,B 0,C 180,E1 32782.178,E2 32782.178} C_VEL
LIN {X 0,Y 720.22,Z 314.513,A -85,B 0,C 180,E1 32779.262,E2 32779.262} C_VEL
LIN {X 0,Y 720.187,Z 314.516,A -85,B 0,C 180,E1 32776.287,E2 32776.287} C_VEL
LIN {X 0,Y 720.22,Z 314.521,A -85,B 0,C 180,E1 32773.406,E2 32773.406} C_VEL
LIN {X 0,Y 720.202,Z 314.51,A -85,B 0,C 180,E1 32770.398,E2 32770.398} C_VEL
LIN {X 0,Y 720.217,Z 314.516,A -85,B 0,C 180,E1 32767.418,E2 32767.418} C_VEL
LIN {X 0,Y 720.217,Z 314.519,A -85,B 0,C 180,E1 32764.299,E2 32764.299} C_VEL
LIN {X 0,Y 720.2,Z 314.51,A -85,B 0,C 180,E1 32761.432,E2 32761.432} C_VEL
LIN {X 0,Y 720.223,Z 314.516,A -85,B 0,C 180,E1 32758.329,E2 32758.329} C_VEL
LIN {X 0,Y 720.192,Z 314.523,A -85,B 0,C 180,E1 32755.425,E2 32755.425} C_VEL
LIN {X 0,Y 720.203,Z 314.509,A -85,B 0,C 180,E1 32752.501,E2 32752.501} C_VEL
LIN {X 0,Y 720.192,Z 314.511,A -85,B 0,C 180,E1 32749.602,E2 32749.602} C_VEL
LIN {X 0,Y 720.191,Z 314.522,A -85,B 0,C 180,E1 32746.839,E2 32746.839} C_VEL
LIN {X 0,Y 720.214,Z 314.52,A -85,B 0,C 180,E1 32743.962,E2 32743.962} C_VEL
LIN {X 0,Y 720.192,Z 314.515,A -85,B 0,C 180,E1 32740.958,E2 32740.958} C_VEL
LIN {X 0,Y 720.232,Z 314.623,A -85,B 0,C 180,E1 32740.475,E2 32740.475} C_VEL
LIN {X 0,Y 721.381,Z 317.779,A -85,B 0,C 180,E1 32740.064,E2 32740.064} C_VEL
LIN {X 0,Y 722.905,Z 320.104,A -85,B 0,C 180,E1 32739.685,E2 32739.685} C_VEL
LIN {X 0,Y 724.843,Z 323.779,A -85,B 0,C 180,E1 32739.151,E2 32739.151} C_VEL
LIN {X 0,Y 730.526,Z 334.884,A -85,B 0,C 180,E1 32737.614,E2 32737.614} C_VEL
LIN {X 0,Y 729.738,Z 367.691,A -85,B 0,C 180,E1 32735.124,E2 32735.124} C_VEL
LIN {X 0,Y 728.84,Z 405.942,A -85,B 0,C 180,E1 32732.374,E2 32732.374} C_VEL
LIN {X 0,Y 727.977,Z 443.258,A -85,B 0,C 180,E1 32729.821,E2 32729.821} C_VEL
LIN {X 0,Y 727.204,Z 482.445,A -85,B 0,C 180,E1 32727.244,E2 32727.244} C_VEL
LIN {X 0,Y 726.727,Z 530.094,A -85,B 0,C 180,E1 32724.214,E2 32724.214} C_VEL
LIN {X 0,Y 728.301,Z 540.273,A -85,B 0,C 180,E1 32723.476,E2 32723.476} C_VEL
LIN {X 0,Y 731.224,Z 547.999,A -85,B 0,C 180,E1 32722.814,E2 32722.814} C_VEL
LIN {X 0,Y 735.504,Z 554.008,A -85,B 0,C 180,E1 32722.185,E2 32722.185} C_VEL
LIN {X 0,Y 738.544,Z 556.698,A -85,B 0,C 180,E1 32721.777,E2 32721.777} C_VEL
LIN {X 0,Y 740.994,Z 557.944,A -85,B 0,C 180,E1 32721.335,E2 32721.335} C_VEL
LIN {X 0,Y 742.745,Z 557.725,A -85,B 0,C 180,E1 32720.84,E2 32720.84} C_VEL
LIN {X 0,Y 743.382,Z 556.189,A -85,B 0,C 180,E1 32720.39,E2 32720.39} C_VEL
LIN {X 0,Y 742.927,Z 553.122,A -85,B 0,C 180,E1 32719.933,E2 32719.933} C_VEL
LIN {X 0,Y 741.37,Z 549,A -85,B 0,C 180,E1 32719.561,E2 32719.561} C_VEL
LIN {X 0,Y 738.792,Z 543.791,A -85,B 0,C 180,E1 32719.278,E2 32719.278} C_VEL
LIN {X 0,Y 734.739,Z 534.807,A -85,B 0,C 180,E1 32719.003,E2 32719.003} C_VEL
LIN {X 0,Y 731.773,Z 524.328,A -85,B 0,C 180,E1 32718.801,E2 32718.801} C_VEL
LIN {X 0,Y 729.965,Z 511.905,A -85,B 0,C 180,E1 32718.677,E2 32718.677} C_VEL
LIN {X 0,Y 729.419,Z 499.525,A -85,B 0,C 180,E1 32718.639,E2 32718.639} C_VEL
LIN {X 0,Y 729.284,Z 327.895,A -85,B 0,C 180,E1 32718.63,E2 32718.63} C_VEL
LIN {X 0,Y 726.568,Z 324.351,A -85,B 0,C 180,E1 32718.441,E2 32718.441} C_VEL
LIN {X 0,Y 723.207,Z 319.856,A -85,B 0,C 180,E1 32718.204,E2 32718.204} C_VEL
